// TwinCAT 3 PLC project PLC
// Title: StateFramework
// Company: RoddenLab
// Author: Kevin Rodden
// ProjectVersion: 1.0.0
// Description: Libary for state-based design of PLC software.
// ProgramVersion: 3.1.4023.0
// libraries:
//   Tc2_Standard, * (Beckhoff Automation GmbH)
//   Tc2_System, * (Beckhoff Automation GmbH)
//   Tc2_TcpIp, * (Beckhoff Automation GmbH)
//   Tc2_Utilities, * (Beckhoff Automation GmbH)
//   Tc3_Module, * (Beckhoff Automation GmbH)
// project tree:
//   DUTs/ ComponentIdentifier.TcDUT, DINT100FIFOBuffer.TcDUT, FaultMessage.TcDUT, Framework.TcDUT, FrameworkLocal.TcDUT, GeneralMessage.TcDUT, HMIBanner.TcDUT, HMIMessage.TcDUT, HMIMessageBuffer.TcDUT, ID50FIFOBuffer.TcDUT, LREAL100FIFOBuffer.TcDUT, StateTimeStamp.TcDUT, Station.TcDUT, TraceFIFOBuffer.TcDUT
//   DUTs/Stats/ Component_Stats.TcDUT, StatsAggregateFIFOBuffer.TcDUT, StatsAggregateRecord.TcDUT, StatsConstants.TcDUT, StatsEvent.TcDUT, StatsEventFIFOBuffer.TcDUT, StatsFailure.TcDUT, StatsFailureFIFOBuffer.TcDUT, StatsFault.TcDUT, StatsFaultFIFOBuffer.TcDUT, StatsShiftAggregateFIFOBuffer.TcDUT, StatsShiftAggregateRecord.TcDUT
//   ENUMs/ eChannel.TcDUT, eColor.TcDUT, eRxMode.TcDUT
//   / PlcTask.TcTTO
//   POUs/Framework/ FB_Framework.TcPOU, FB_StationState.TcPOU, FIFO_HMIMessage.TcPOU, F_FindMessage.TcPOU, FB_StationControl.TcPOU
//   POUs/OEE/ FIFO_StatsAggregate.TcPOU, FIFO_StatsEvent.TcPOU, FIFO_StatsFailureLog.TcPOU, FIFO_StatsFaultLog.TcPOU, FIFO_StatsShiftAggregate.TcPOU, F_SendEvent.TcPOU
//   POUs/Serial Communication/ FB_EL6001.TcPOU, FB_EL6002.TcPOU
//   POUs/State Trace/ FIFO_StateTrace.TcPOU
//   POUs/TCP Communication/ FB_TCPClient.TcPOU
//   POUs/Utility/ FB_Blinker.TcPOU, FB_FileReadSettings.TcPOU, FB_FileWriteSettings.TcPOU, FB_Sensor.TcPOU, FIFO_DINT100.TcPOU, FIFO_ID50.TcPOU, FIFO_LREAL100.TcPOU, F_GetTimeStamp.TcPOU, LEFTBigString.TcPOU, RIGHTBigString.TcPOU
// real-time tasks:
//   TASK PlcTask: cycle T#10ms, priority 20, ADS port 350

CONFIGURATION PLC
    RESOURCE PLC ON TwinCAT3
        TASK PlcTask(INTERVAL := T#10ms, PRIORITY := 20);
    END_RESOURCE
END_CONFIGURATION

// ---- DUTs/ComponentIdentifier.TcDUT
TYPE ComponentIdentifier :
STRUCT
	ID		: DINT;		// Component ID
	Name	: STRING;	// Component Name
END_STRUCT
END_TYPE

// ---- DUTs/DINT100FIFOBuffer.TcDUT
TYPE DINT100FIFOBuffer :
STRUCT
	Size	: UDINT := 100;				// Size of FIFO
	Buffer	: ARRAY [0..99] OF DINT;	// Buffer of FIFO Elements
END_STRUCT
END_TYPE

// ---- DUTs/FaultMessage.TcDUT
TYPE FaultMessage :
STRUCT
	Id		: DINT;			// Identifier for Fault Condition
	Text	: T_MaxString;	// Text (Message) for Fault Condition
	AltText	: T_MaxString;	// Alt Text for Fault Condition
END_STRUCT
END_TYPE

// ---- DUTs/Framework.TcDUT
TYPE Framework :
STRUCT
	ComponentIDRecord	: ComponentIdentifier;	// Component Identifier
	Behavior			: DINT;					// Component Behavior Modifier
	OnScan				: BOOL;
	ResetStart			: BOOL;
	ResetDone			: BOOL;
	FullInitRequired	: BOOL;
	EnableStateTrace	: BOOL;
END_STRUCT
END_TYPE

// ---- DUTs/FrameworkLocal.TcDUT
TYPE FrameworkLocal :
STRUCT
	AsynchFault					: BOOL;
	AsynchFaultReactionComplete	: BOOL;
	Attention					: BOOL;
	CycleAuto					: BOOL;
	CycleFaulted				: BOOL;
	CycleManual					: BOOL;
	CycleReset					: BOOL;
	ManualCycleRequested		: BOOL;
	ManualCycleDone				: BOOL;
	OKToStop					: BOOL;
	SingleStepInhibit			: BOOL;
	IgnoreSingleStep			: BOOL;
	FirstEntry					: BOOL;
	LongFaultState				: BOOL;
	CycleAutoFallingEdge		: F_TRIG;
	CycleResetFallingEdge		: F_TRIG;
	CycleManualFallingEdge		: F_TRIG;
	State						: DINT;
	NextState					: DINT;
	LastAutoState				: DINT;
	ReEntryState				: DINT;
	FaultedState				: DINT;
	FaultNumber					: DINT;
	LocalFaultID				: DINT;
	FullFaultID					: DINT;
	tmrState					: TON;
	tmrFault					: TON;
	StateTimePreset				: TIME;
	FaultTimePreset				: TIME;
	FaultTimeLong				: TIME;
	FaultTimeShort				: TIME;
	FaultText					: T_MaxString;
	FaultAltText				: T_MaxString;
	FaultData					: StatsFault;
	MsgText						: T_MaxString;
	AltMsgText					: T_MaxString;
	MsgArray					: ARRAY [0..99] OF GeneralMessage;
	HMIMsg						: HMIMessage;
	StateTimeStamp				: StateTimeStamp;
	CurrentTime					: TimeStamp;
	Name						: STRING(30);
	AltName						: STRING(30);
	pStateTraceBuffer			: POINTER TO TraceFIFOBuffer;
	pStateTraceFifo				: POINTER TO FIFO_StateTrace;
	pStats						: POINTER TO Component_Stats;
END_STRUCT
END_TYPE

// ---- DUTs/GeneralMessage.TcDUT
TYPE GeneralMessage :
STRUCT
	Id: DINT;
	BitNumber: DINT;
	Text: STRING;
	AltText: STRING;
END_STRUCT
END_TYPE

// ---- DUTs/HMIBanner.TcDUT
// HMI Banner Structure Relaying Data to HMI Controls
TYPE HMIBanner :
STRUCT
	Text	: T_MaxString;	// Text for HMI Banner
	AltText	: T_MaxString;	// Additional Text for HMI Banner
	Color	: eColor;		// Color of HMI Banner Background
END_STRUCT
END_TYPE

// ---- DUTs/HMIMessage.TcDUT
TYPE HMIMessage :
STRUCT
	Channel	: eChannel;		// Channel for HMI Message
	Color	: eColor;		// Color of HMI Message (Background)
	Text	: T_MaxString;	// Text of HMI Message
	AltText	: T_MaxString;	// Additional Text for HMI Message
END_STRUCT
END_TYPE

// ---- DUTs/HMIMessageBuffer.TcDUT
TYPE HMIMessageBuffer :
STRUCT
	Size	: UDINT := 100;					// Array Size for HMI Message FIFO Buffer
	Buffer	: ARRAY [0..99] OF HMIMessage;	// FIFO Buffer for HMI Messages 
END_STRUCT
END_TYPE

// ---- DUTs/ID50FIFOBuffer.TcDUT
TYPE ID50FIFOBuffer :
STRUCT
	Size: UDINT := 50;
	Buffer: ARRAY [0..49] OF ComponentIdentifier;
END_STRUCT
END_TYPE

// ---- DUTs/LREAL100FIFOBuffer.TcDUT
TYPE LREAL100FIFOBuffer :
STRUCT
	Size: UDINT := 100;
	Buffer: ARRAY [0..99] OF LREAL;
END_STRUCT
END_TYPE

// ---- DUTs/StateTimeStamp.TcDUT
TYPE StateTimeStamp :
STRUCT
	Station		: DINT;	
	ID			: DINT;
	State		: DINT;
	DateTime	: TIMESTRUCT;
END_STRUCT
END_TYPE

// ---- DUTs/Station.TcDUT
TYPE Station :
STRUCT
	FirstScan					: BOOL	:= TRUE;	// First Scan for PLC Startup
	
	CycleAuto					: BOOL;					// Flag Indicating 
	CycleReset					: BOOL;
	CycleManual					: BOOL;
	CycleStopped				: BOOL;
	CycleFaulted				: BOOL;
	
	OKToStart					: BOOL;					// Flag Indicating Station Readiness to Start Cycling
	OKToStop					: BOOL;					// Flag Indicating Station Readiness to Stop Cycling
	OKToReset					: BOOL;					// Flag Indicating Station Readiness to Reset Faults/Handshakes
	OKForManual					: BOOL;					// Flag Indicating Station Readiness to Enter Manual Mode
	
	StopRequest					: BOOL;
	EmergencyStop				: BOOL;
	UnlatchFaults				: BOOL;
	FaultReset					: BOOL;
	StationResetRequired		: BOOL;					// Flag Indicating Full Station Reset Required
	ResetDone					: BOOL;
	SingleStep					: BOOL;
	StepAdvance					: BOOL;
	DryCycle					: BOOL;
	Attention					: BOOL;
	MachineStopRequest			: BOOL;
	StationID					: DINT;					// Identifier for the Station
	
	FirstFault					: StatsFault;			
	UpstreamStationID			: DINT;					// Upstream Station Identifier
	DownstreamStationID			: DINT;					// Downstream Station Identifier
	
	StationMessage				: HMIBanner;
	OperatorMessage				: HMIBanner;
	b500msPulse					: BOOL;					// Global 500ms Boolean Pulse

	FaultedFIFO					: FIFO_ID50;			// FIFO of Faulted Components
	FaultedFIFOBuffer			: ID50FIFOBuffer;		// Faulted Component FIFO Memory
	
	NotOKtoStopFIFO				: FIFO_ID50;			// FIFO of Not OK to Stop Components
	NotOKToStopFIFOBuffer		: ID50FIFOBuffer;		// Not OK to Stop FIFO Memory
	
	HMIMessageFIFO				: FIFO_HMIMessage;		// FIFO of HMI Messages
	HMIMessageBuffer			: HMIMessageBuffer;		// HMI Message FIFO Memory
	
	AttentionRequiredFIFO		: FIFO_ID50;			// FIFO of Components Requiring Attention
	AttentionRequiredFIFOBuffer	: ID50FIFOBuffer;		// Attention Request FIFO Memory
	
	CycleManualFIFO				: FIFO_ID50;
	CycleManualFIFOBuffer		: ID50FIFOBuffer;
	
	StationStateTraceFifo		: FIFO_StateTrace;
	StationStateTraceBuffer		: TraceFIFOBuffer;	
END_STRUCT
END_TYPE

// ---- DUTs/Stats/Component_Stats.TcDUT
TYPE Component_Stats :
STRUCT
	AggregateInterval			: DINT; 						(*interval time in minutes*)
	PlannedDowntime				: ARRAY [0..2] OF DINT;  		(*index corresponds to shift number*)
	StartOfShift				: ARRAY [0..2, 0..1] OF DINT; 	(*[shift number],[hour,min]*)
	IdealCycleTime				: LREAL; 						(*cycle time is second*)
	StatsEventFIFO				: FIFO_StatsEvent 			:= (Overwrite := TRUE);
	StatsEventBuffer			: StatsEventFIFObuffer;
	StatsAggregateFIFO			: FIFO_StatsAggregate 		:= (Overwrite := TRUE);
	StatsAggregateBuffer		: StatsAggregateFIFOBuffer;
	StatsShiftAggregateFIFO		: FIFO_StatsShiftAggregate 	:= (Overwrite := TRUE);
	StatsShiftAggregateBuffer	: StatsShiftAggregateFIFOBuffer;
	StatsFaultLog				: FIFO_StatsFaultLog 		:= (Overwrite := TRUE);
	StatsFaultLogBuffer			: StatsFaultFIFOBuffer;
	StatsFailureLog				: FIFO_StatsFailureLog 		:= (Overwrite := TRUE);
	StatsFailureLogBuffer		: StatsFailureFIFOBuffer;
	StatsIdealCycleTimeFIFO		: FIFO_LREAL100;
	StatsIdealCycleTimeBuffer	: LREAL100FIFOBuffer;
	StatsPartCountFIFO			: FIFO_DINT100;
	StatsPartCountBuffer		: DINT100FIFOBuffer;
	Framework					: Framework;
END_STRUCT
END_TYPE

// ---- DUTs/Stats/StatsAggregateFIFOBuffer.TcDUT
TYPE StatsAggregateFIFOBuffer :
STRUCT
	Size: UDINT := 864; (*3 days at 5 min*)
	Buffer: ARRAY [0..863] OF StatsAggregateRecord;
END_STRUCT
END_TYPE

// ---- DUTs/Stats/StatsAggregateRecord.TcDUT
TYPE StatsAggregateRecord :
STRUCT
	TimeStamp: TimeStamp;
	OperatorStopTime: LREAL;
	OperatorStopCount: DINT;
	AutoStopTime: LREAL;
	AutoStopCount: DINT;
	WorkTime: LREAL;
	WorkCount: DINT;
	BypassTime: LREAL;
	BypassCount: DINT;
	BlockTime: LREAL;
	BlockCount: DINT;
	StarveTime: LREAL;
	StarveCount: DINT;
	FaultTime: LREAL;
	FaultCount: DINT;
	EmptyTime: LREAL;
	EmptyCount: DINT;
	RetryTime: LREAL;
	RetryCount: DINT;
	MasterTime: LREAL;
	MasterCount: DINT;
	OtherTime: LREAL;
	OtherCount: DINT;
	RejectCount: DINT;
	GoodCount: DINT;
	FirstTimeGoodCount: DINT;
	FirstTimeStartCount: DINT;
	GoodCycleTime: LREAL;
	InitCount: DINT;
	PartsForCurrentCycleTime: DINT;
	Shift: DINT;
END_STRUCT
END_TYPE

// ---- DUTs/Stats/StatsConstants.TcDUT
TYPE StatsConstants :
STRUCT
	Aggregate: DINT := 1;

	OperatorStop: DINT := 100;
	MachineStop: DINT := 101;
	Working: DINT := 102;
	Bypass: DINT := 103;
	Blocked: DINT := 104;
	Starved: DINT := 105;
	Faulted: DINT := 106;
	FaultAcknowledge: DINT := 107;
	Empty: DINT := 108;
	Retry: DINT := 109;
	Mastering: DINT := 110;

	Failure: DINT := 200;
	Good: DINT := 201;
	FirstTimeGood: DINT := 202;
	FirstTimeStart: DINT := 203;
	Initialize: DINT := 204;

	PartChange: DINT := 300;
	CycleTime: DINT := 301;
END_STRUCT
END_TYPE

// ---- DUTs/Stats/StatsEvent.TcDUT
TYPE StatsEvent :
STRUCT
	TimeStamp: TimeStamp;
	EType: DINT;
	Data: ARRAY [0..4] OF REAL;
	StringData: ARRAY [0..3] OF STRING;
END_STRUCT
END_TYPE

// ---- DUTs/Stats/StatsEventFIFOBuffer.TcDUT
TYPE StatsEventFIFOBuffer :
STRUCT
	Size: UDINT := 100;
	Buffer: ARRAY [0..99] OF StatsEvent;
END_STRUCT
END_TYPE

// ---- DUTs/Stats/StatsFailure.TcDUT
TYPE StatsFailure :
STRUCT
	TimeStamp: TimeStamp;
	StationID: DINT;
	FailureID: DINT;
	Parameters: STRING;
END_STRUCT
END_TYPE

// ---- DUTs/Stats/StatsFailureFIFOBuffer.TcDUT
TYPE StatsFailureFIFOBuffer :
STRUCT
	Size: UDINT := 500;
	Buffer: ARRAY [0..499] OF StatsFailure;
END_STRUCT
END_TYPE

// ---- DUTs/Stats/StatsFault.TcDUT
TYPE StatsFault:
STRUCT
	TimeStamp: TimeStamp;
	StationID: DINT;
	FaultID: DINT;
	AcknowledgeTime: LREAL;
	Duration: LREAL;
	Data: ARRAY [0..2] OF REAL;
	StringData: ARRAY [0..3] OF STRING;
END_STRUCT
END_TYPE

// ---- DUTs/Stats/StatsFaultFIFOBuffer.TcDUT
TYPE StatsFaultFIFOBuffer :
STRUCT
	Size: UDINT := 500;
	Buffer: ARRAY [0..499] OF StatsFault;
END_STRUCT
END_TYPE

// ---- DUTs/Stats/StatsShiftAggregateFIFOBuffer.TcDUT
TYPE StatsShiftAggregateFIFOBuffer :
STRUCT
	Size: UDINT := 270; (*90 days*)
	Buffer: ARRAY [0..269] OF StatsShiftAggregateRecord;
END_STRUCT
END_TYPE

// ---- DUTs/Stats/StatsShiftAggregateRecord.TcDUT
TYPE StatsShiftAggregateRecord :
STRUCT
	AggregateData: StatsAggregateRecord;
	Shift: DINT;
	ShiftStartTimeStamp: TimeStamp;
	AvailableTime: LREAL;
	NetAvailableTime: LREAL;
	TotalDownTime: LREAL;
	PlannedDownTime: LREAL;
	UnplannedDownTime: LREAL;
	OperatingTime: LREAL;
	EquipmentAvailability: LREAL;
	TotalParts: DINT;
	PerformanceEfficiency: LREAL;
	QualityRate: LREAL;
	OverallEquipmentEffectiveness: LREAL;
	CycleTimeAvgSum: LREAL;
	CycleTimeAvgCnt: DINT;
END_STRUCT
END_TYPE

// ---- DUTs/TraceFIFOBuffer.TcDUT
TYPE TraceFIFOBuffer :
STRUCT
	Size: UDINT := 1000;
	Buffer: ARRAY [0..999] OF StateTimeStamp;
END_STRUCT
END_TYPE

// ---- ENUMs/eChannel.TcDUT
{attribute 'qualified_only'}
{attribute 'strict'}
TYPE eChannel :
(
	Unspecified	:= 0,	// Message Channel Not Defined
	Fault 		:= 1,	// Fault Channel
	Attention 	:= 2,	// Attention Required Channel
	General 	:= 3,	// General Information Channel
	FirstFault 	:= 4	// First Fault (Startup) Channel
) DINT := Unspecified;
END_TYPE

// ---- ENUMs/eColor.TcDUT
{attribute 'qualified_only'}
{attribute 'strict'}
TYPE eColor :
(
	Black 	:= 16#000000,	// Black RGB Code
	Red	 	:= 16#FF0000,	// Red RGB Code
	Green 	:= 16#00FF00,	// Green RGB Codde
	Blue 	:= 16#0000FF,	// Blue RGB Codee
	Grey 	:= 16#F2F2F2,	// Gray RGB Code
	Yellow 	:= 16#FFFF00,	// Yellow RGB Code
	White 	:= 16#FFFFFF	// White RGB Code
) DINT := Black;
END_TYPE

// ---- ENUMs/eRxMode.TcDUT
{attribute 'qualified_only'}
{attribute 'strict'}
TYPE eRxMode :
(
	Delimited	:= 0,
	FixedLength := 1,
	Continuous	:= 2
);
END_TYPE

// ---- POUs/Framework/FB_Framework.TcPOU
FUNCTION_BLOCK FB_Framework
VAR_INPUT
	ComponentIDRecord	: ComponentIdentifier;	// Information to Identify Component
	CurrentTime			: TimeStamp;			// Current System Time
END_VAR

VAR_IN_OUT
	Local				: FrameworkLocal;		// Framework Local Structure Reference
	Station				: Station;				// Station Object Reference
END_VAR

VAR
	Message				: GeneralMessage;		// Fault Message Memory Buffer
	HMIMessage			: HMIMessage;			// HMI Message Memory Buffer		
END_VAR

// Initialize Framework Local Fields
IF Station.FirstScan THEN
	Local.State 		:= 9999;
	Local.NextState 	:= 5000;
	Local.FaultedState 	:= 0;
	Local.ReEntryState 	:= 0;
	Local.LastAutoState := 0;
	Local.FaultNumber 	:= 0;
END_IF

(****************************************************************************
* Framework Post-Sequence Logic, DO NOT modify this section *
*****************************************************************************)

(****************************************************************************
* State Timeout Fault Logic *
*****************************************************************************)
// Set the State Fault Timer to Preset 
Local.tmrFault(PT := Local.FaultTimePreset);

// If Component in Auto, Reset, or Manual, Fault Enabled
IF Local.CycleAuto OR Local.CycleReset OR Local.CycleManual THEN
	// If Component OK to Stop or Single Stepping, Fault Disabled
	IF NOT Local.OKToStop AND NOT Station.SingleStep THEN
		// If State Stuck for Duration, Trigger Fault
		Local.tmrFault(IN := Local.NextState = Local.State);
	ELSE
		Local.tmrFault(IN := FALSE);
	END_IF
ELSE
	Local.tmrFault(IN := FALSE);
END_IF

// Unlatch Fault Condition When Directed by Station
IF Station.UnlatchFaults THEN
	Local.CycleFaulted := FALSE;
	Local.FaultNumber := 0;
END_IF

// Check if Fault Condition Present
IF Local.FaultNumber > 0 THEN
	
	// If Component not Faulted, Trigger Fault Condition
	IF NOT Local.CycleFaulted THEN
		Local.CycleFaulted := TRUE;
	
		// Check if Fault Occured in Sync with State Machine
		// Set Faulted State/FaultID Accordingly
		IF NOT Local.AsynchFault OR Local.AsynchFaultReactionComplete THEN
			Local.FaultedState := Local.State;
			Local.LocalFaultID := Local.FaultedState * 10 + Local.FaultNumber; // Faulted State Used in Identifier
		ELSE
			Local.FaultedState := 0;
			Local.LocalFaultID := Local.FaultNumber; // No Faulted State Included (Async == Global in this case)
		END_IF
		
		// Set Full Fault ID (Includes Component ID)
		Local.FullFaultID := ComponentIDRecord.ID * 100000 + Local.LocalFaultID;
		Local.FaultData.FaultID := Local.FullFaultID;
		
		// Fetch Message for Fault Condition
		Message := F_FindMessage(Local.MsgArray, Local.FaultedState, Local.FaultNumber);
		
		// Set Local Fault Message Text
		Local.MsgText := 'Fault: ';
		Local.MsgText := CONCAT(Local.MsgText, DINT_TO_STRING(Local.FaultData.FaultID));
		Local.MsgText := CONCAT(Local.MsgText, ' ');
		Local.MsgText := CONCAT(Local.MsgText, Local.Name);
		Local.MsgText := CONCAT(Local.MsgText, ' - ');
		Local.MsgText := CONCAT(Local.MsgText, Message.Text);
		
		// Set Local Alt Fault Message Text
		Local.AltMsgText := 'AltFault: ';
		Local.AltMsgText := CONCAT(Local.AltMsgText, DINT_TO_STRING(Local.FaultData.FaultID));
		Local.AltMsgText := CONCAT(Local.AltMsgText, ' ');
		Local.AltMsgText := CONCAT(Local.AltMsgText, Local.AltName);
		Local.AltMsgText := CONCAT(Local.MsgText, ' - ');
		Local.AltMsgText := CONCAT(Local.AltMsgText, Message.AltText);
		
		// Add Message to Station Buffer
		HMIMessage.Text		:= Message.Text;
		HMIMessage.AltText 	:= Message.AltText;
		HMIMessage.Channel	:= eChannel.Fault;
		HMIMessage.Color	:= eColor.Red;
		Station.HMIMessageFIFO.LOAD(HMIMessage := HMIMessage);
		
		// Check if Component Fault Already Active
		// Set Station First Fault to Current Fault if Not Active
		IF Station.FirstFault.FaultID = 0 THEN
			Station.FirstFault 					:= Local.FaultData;
			Station.FirstFault.StationID 		:= Station.StationID;
			Station.FirstFault.StringData[0] 	:= Local.MsgText;
			Station.FirstFault.StringData[1] 	:= Local.AltMsgText;
			Station.FirstFault.StringData[2] 	:= Local.FaultData.StringData[2];
			Station.FirstFault.Data 			:= Local.FaultData.Data;
		END_IF
	END_IF
END_IF


// If Cycle Faulted, Load Fault to FIFO
IF Local.CycleFaulted THEN
	Station.FaultedFIFO.LOAD(pFIFO := ADR(Station.FaultedFIFOBuffer), In := ComponentIDRecord);
END_IF

// If Cycle Manual, Load Manual to FIFO
IF Local.CycleManual THEN
	Station.CycleManualFIFO.LOAD(pFIFO := ADR(Station.CycleManualFIFOBuffer), in := ComponentIDRecord);
END_IF

// If Attention Flagged, Load to Station FIFO
IF Local.Attention THEN
	Station.AttentionRequiredFIFO.LOAD(pFIFO := ADR(Station.AttentionRequiredFIFOBuffer), in := ComponentIDRecord);
END_IF

// If Not OK to Stop, Load to Station FIFO
IF NOT Local.OKToStop AND NOT Local.CycleFaulted THEN
	Station.NotOKtoStopFIFO.LOAD(pFIFO := ADR(Station.NotOKtoStopFIFOBuffer), in := ComponentIDRecord);
END_IF


(***************************************************************************
* Framework Pre-Sequence Logic, DO NOT modify this section *
****************************************************************************)

// Set Cycle Auto if Station in Auto and Component Not Faulted
Local.CycleAuto := Station.CycleAuto AND NOT Local.CycleFaulted;

// Set Cycle Reset if Station in Reset and Component Not Faulted
Local.CycleReset := Station.CycleReset AND NOT Local.CycleFaulted;

// Set Cycle Manual if Component Requesting Manual and Station Not Faulted
Local.CycleManual := Local.ManualCycleRequested AND NOT Local.ManualCycleDone AND NOT Station.CycleFaulted;

// Set Single Step Mode if Station in Single Step (not Advancing) and Component Enabled
Local.SingleStepInhibit := Station.SingleStep AND NOT Station.StepAdvance AND NOT Local.IgnoreSingleStep;



(*On the falling edge of CycleAuto, grab the current state as LastAutoState.
Also, set the default ReEntryState to the LastAutoState so that we pick back up where we left off after a simple cycle stop / cycle start.
Set State to 5000, the Idle state.
Note that we block the capture of LastAutoState and setting of ReEntryState if we are currently in states 5000 or 5001.
This is to avoid overwriting these values in the rare case that an AsynchFault occurs in the same scans that we are
transitioning out of 5000, or while in 5001.*)
Local.CycleAutoFallingEdge(CLK:=Local.CycleAuto);
IF Local.CycleAutoFallingEdge.Q THEN
	IF Local.State <> 5000 AND Local.State <> 5001 THEN
		Local.LastAutoState := Local.State;
		Local.ReEntryState := Local.LastAutoState;
	END_IF
	Local.NextState := 5000;
END_IF

// On Cycle Reset Falling Edge, Set State to 5000 (Idle)
Local.CycleResetFallingEdge(CLK := Local.CycleReset);
IF Local.CycleResetFallingEdge.Q THEN
	Local.NextState := 5000;
END_IF

// On Manual Cycle Falling Edge, Set State to 5000
Local.CycleManualFallingEdge(Clk:=Local.CycleManual);
IF Local.CycleManualFallingEdge.Q THEN
	Local.NextState := 5000;
END_IF

// On State Transition
IF Local.NextState <> Local.State THEN
	// Set First Entry Flag
	Local.FirstEntry := TRUE;
	
	// Set State Equal to Next State (Update)
	Local.State := Local.NextState;
	
	// Update Current Time
	Local.CurrentTime := CurrentTime;
	
	// Set Data for State Trace Buffer
	Local.StateTimeStamp.ID := ComponentIDRecord.ID;
	Local.StateTimeStamp.State := Local.State;
	Local.StateTimeStamp.DateTime := Local.CurrentTime;
	
	// Add Entry to State Trace Buffer
	Local.pStateTraceFifo^.LOAD(pFIFO := Local.pStateTraceBuffer, IN := Local.StateTimeStamp);
	
ELSE
	// Reset First Entry Flag
	Local.FirstEntry := FALSE;
	
END_IF

// State Idle Timer
Local.tmrState(
	IN := Local.NextState = Local.State,
	PT := Local.StateTimePreset);

// Reset OK to Stop Condition
Local.OKToStop := FALSE;

END_FUNCTION_BLOCK

// ---- POUs/Framework/F_FindMessage.TcPOU
// Function to Retrieve Message from Provided Buffer Mapped to the Provided State/ID Combination
FUNCTION F_FindMessage : GeneralMessage

VAR_INPUT
	MessageArray	: ARRAY [0..99] OF GeneralMessage;	// Array of Messages
	State			: DINT;								// State Reference 
	ID				: DINT;								// Fault ID Reference
END_VAR

VAR
	Message			: GeneralMessage;					// Temporary Message Buffer
	Index			: DINT;								// Index for Array Search
	Length			: DINT;								// Number of Array Elements
END_VAR

// Get Length of Message Array
Length := SIZEOF(MessageArray) / SIZEOF(Message);

// Set Message Text to Defaults
Message.Text 	:= '**No message text**';
Message.AltText := '**No alt message text**';

// Search Message Array for Fault Message
FOR Index := 0 TO (length - 1) DO
	// If Message ID Matches State ID, Set Message Buffer to Array Element
	IF MessageArray[Index].Id = (State * 10 + ID) THEN
		Message := MessageArray[Index];
		EXIT;
	END_IF
END_FOR

// Set Output to Message Buffer
F_FindMessage := Message;

END_FUNCTION

// ---- POUs/Framework/FB_StationState.TcPOU
FUNCTION_BLOCK FB_StationState
// Station State Commands
VAR_INPUT
	StationResetCommand		: BOOL;
	FaultAcknowledgeCommand	: BOOL;
	FaultResetCommand		: BOOL;
	StationLevelFault		: BOOL;
	CycleStartCommand		: BOOL;
	CycleStopCommand		: BOOL;
	ManualModeCommand		: BOOL;
END_VAR

// Configuration Inputs
VAR_INPUT
	SeperateAckAndReset		: BOOL;		// Configuration to Require Fault Acknowledge
	ResetAfterManualMode	: BOOL;		// Configuration to Require Station Reset After Leaving Manual Mode
END_VAR

VAR_IN_OUT
	Station					: Station;
END_VAR

VAR_OUTPUT
	StationStateMessage		: T_MaxString;
END_VAR

VAR
	State					: DINT;
	NextState				: DINT;
	FirstEntry				: BOOL;
	WaitForFaultAck			: BOOL;
	CurrentTime				: TIMESTRUCT;
	ModeTimeStamp			: StateTimeStamp;
END_VAR

// First Scan
IF Station.FirstScan THEN
	State 		:= 9999;
	NextState 	:= 0;
END_IF


// Async Setting for Init Required Flag
IF StationResetCommand THEN
	Station.StationResetRequired := TRUE;
END_IF;


// Mode Control State Machine
CASE State OF
		
	0:	// Faulted, Not Acknowledged
	
		StationStateMessage := 'Faulted, Not Acknowledged';
	
		IF FaultAcknowledgeCommand OR NOT SeperateAckAndReset THEN
			FaultAcknowledgeCommand := FALSE;
			NextState := 10;
		END_IF;
		
	
	10:	// Faulted, Acknowledged
	
		IF FirstEntry THEN
			IF SeperateAckAndReset THEN
				StationStateMessage := 'Fault Acknowledged';
			END_IF;
			WaitForFaultAck := TRUE;
		END_IF;
	
		// Check if Station Ready for Reset
		IF Station.OKToReset THEN
			
			IF WaitForFaultAck AND SeperateAckAndReset THEN
				WaitForFaultAck := FALSE;
				
				IF Station.StationResetRequired THEN
					StationStateMessage := 'Waiting for Station Reset';
				ELSE
					StationStateMessage := 'Waiting for Station or Fault Reset';
				END_IF
			END_IF;
			
			// Check if Station Reset Required
			IF Station.StationResetRequired THEN
				
				// Station Reset Commanded
				IF StationResetCommand THEN
					StationResetCommand 		:= FALSE;
					NextState 			:= 50;
					Station.SingleStep	:= FALSE;
				END_IF
				
				// Fault Reset - Reject
				IF FaultResetCommand THEN
					StationStateMessage := 'Station Reset Required'; 
				END_IF
				
			ELSE
				// Station Reset Commanded
				IF StationResetCommand THEN
					StationResetCommand 		:= FALSE;
					NextState 			:= 50;
					Station.SingleStep	:= FALSE;
				END_IF;
			
				// Fault Reset Commanded
				IF FaultResetCommand THEN
					FaultResetCommand 			:= FALSE;
					NextState  			:= 20;
					Station.SingleStep	:= FALSE;
				END_IF;
			END_IF
			
		END_IF;
		
	
	20	:	// Unlatch Faults, Fault Reset
	
		IF FirstEntry THEN
			Station.UnlatchFaults := TRUE;
			StationStateMessage := 'Unlatching Faults...';
		END_IF;
	
		IF NOT Station.CycleFaulted AND NOT StationLevelFault THEN
			NextState	:= 30;
		END_IF;
	
		IF NextState <> State THEN
			Station.UnlatchFaults := FALSE;
		END_IF
		
		
	30:	// Fault Reset
	
		// Command Component Reset 
		IF FirstEntry THEN
			Station.CycleReset 	:= TRUE;
			StationStateMessage 		:= 'Resetting...';
		END_IF;
	
		// Wait for Reset Complete
		IF Station.ResetDone THEN
			NextState := 100;
		END_IF;
		
		// If Station Faults During Reset or Station Reset Commanded, Return to Faulted
		IF Station.CycleFaulted OR StationResetCommand THEN
			StationResetCommand 	:= FALSE;
			NextState 		:= 0;
		END_IF;
		
		// Reset Component Reset
		IF NextState <> State THEN
			Station.CycleReset := FALSE;
		END_IF
		
	
	50	:	// Unlatch Faults - Station Reset*)
	
		// Unlatch Component Faults
		IF FirstEntry THEN
			Station.UnlatchFaults 	:= TRUE;
			StationStateMessage 			:= 'Unlatching Faults...';
		END_IF;
		
		// Wait for Faults (and Station Faults) to Clear
		IF NOT Station.CycleFaulted AND NOT StationLevelFault THEN
			NextState 	:= 60;
		END_IF;
	
		// Reset Fault Unlatch Command
		IF NextState <> State THEN
			Station.UnlatchFaults	:= FALSE;
		END_IF
		
		
	60	:	// Station Reset
	
		// Command Component Resets
		IF FirstEntry THEN
			Station.CycleReset 	:= TRUE;
			StationStateMessage 		:= 'Resetting...';
		END_IF;
	
		// Wait for Component Reset Complete
		IF Station.ResetDone THEN
			Station.StationResetRequired 	:= FALSE;
			NextState 						:= 100;
		END_IF;
		
		// If Fault During Reset, Return to Faulted State
		IF Station.CycleFaulted THEN
			NextState 	:= 0;
		END_IF;
		
		// Reset Component Reset Command on Exit
		IF NextState <> State THEN
			Station.CycleReset := FALSE;
		END_IF
	
		
	100:	// Idle
	
		IF FirstEntry THEN
			StationStateMessage := 'Idle';
		END_IF
	
		// Cycle Start Commanded
		IF CycleStartCommand AND Station.OKToStart THEN
			CycleStartCommand	:= FALSE;
			NextState 	:= 200;
		END_IF
	
		// Manual Mode Commanded
		IF ManualModeCommand AND Station.OKForManual THEN
			ManualModeCommand	:= FALSE;
			NextState	:= 300;
		END_IF
		
		// In Case of Cycle Fault
		IF Station.CycleFaulted THEN
			NextState := 0;
		END_IF;
		
		// Station Reset Commanded
		IF StationResetCommand AND Station.OKToReset THEN
			NextState := 60;
		END_IF
		
	
	200	:	// Running
	
		IF FirstEntry THEN
			Station.CycleAuto 	:= TRUE;
			StationStateMessage 		:= 'Running';
		END_IF
		
		// Cycle Stop, Operator Stop
		IF CycleStopCommand OR Station.CycleFaulted THEN
			CycleStopCommand	:= FALSE;
			NextState 	:= 250;
		END_IF
	
		
	250 :	// Stop Station
	
		IF FirstEntry THEN
			Station.StopRequest := TRUE;
			StationStateMessage 		:= 'Stopping...';
		END_IF;
		
		// Wait for OK To Stop
		IF Station.OKToStop THEN
			Station.StopRequest := FALSE;
			Station.CycleAuto 	:= FALSE;
			// Check if Fault Occured
			IF Station.CycleFaulted THEN
				NextState := 0;
			ELSE
				NextState := 100;
			END_IF
		END_IF
		
		
	300	:	// Manual Mode
	
		IF FirstEntry THEN
			Station.CycleManual := TRUE;
			StationStateMessage 		:= 'Manual Mode';
		END_IF
		
		// Wait for Stop Command or Fault
		IF CycleStopCommand OR Station.CycleFaulted THEN
			CycleStopCommand := FALSE;
			NextState := 250;
		END_IF
		
		IF State <> NextState THEN
			Station.CycleManual				:= FALSE;
			// Set Station Reset if Configured
			Station.StationResetRequired	:= ResetAfterManualMode;
		END_IF
	
END_CASE


// State Update Logic
IF NextState <> State THEN
	FirstEntry 				:= TRUE;
	State 					:= NextState;
	
	// Update State Trace
	ModeTimeStamp.DateTime	:= F_GetTimeStamp();
	ModeTimeStamp.State		:= NextState;
	ModeTimeStamp.Station	:= Station.StationID;
	Station.StationStateTraceFIFO.LOAD(IN := ModeTimeStamp);
ELSE
	FirstEntry 	:= FALSE;
	
END_IF

END_FUNCTION_BLOCK

// ---- POUs/Utility/F_GetTimeStamp.TcPOU
FUNCTION F_GetTimeStamp : TIMESTRUCT
VAR
	fbGetTime		: GETSYSTEMTIME;	// Function Block to Fetch System Time
	TimeStamp		: T_FileTime;		// Time Stamp Structure
	Time64			: T_ULarge_Integer;	// 64-Bit Large Integer Time
	TimeShift		: LREAL;			// Amount for Time Zone Offset Shift 
	TimeZoneOffset	: DINT;				// UTC Time Zone Offset
END_VAR

// Trigger TwinCAT Function Block
fbGetTime(
	timeLoDW => Time64.dwLowPart, 
	timeHiDW => Time64.dwHighPart);

// Correct for Timezone Offset
TimeShift := DINT_TO_LREAL(ABS(TimeZoneOffset)) (*hours*) * DINT_TO_LREAL(3600) (*seconds*) * DINT_TO_LREAL(10000000) (*100ns*);

IF TimeZoneOffset < 0 THEN
	Time64 := UInt64Sub64(Time64, LREAL_TO_UINT64(TimeShift));
ELSE
	Time64 := UInt64Add64(Time64, LREAL_TO_UINT64(TimeShift));
END_IF

// Unpack Large Integer Time
TimeStamp.dwLowDateTime  := Time64.dwLowPart;
TimeStamp.dwHighDateTime := Time64.dwHighPart;

// Unpack TimeStamp to Time Structure
F_GetTimeStamp :=  FILETIME_TO_SYSTEMTIME(TimeStamp);

END_FUNCTION

// ---- POUs/Framework/FIFO_HMIMessage.TcPOU
// HMI Message FIFO
FUNCTION_BLOCK FIFO_HMIMessage

VAR_INPUT
	Overwrite	: BOOL;							// Flag to Overwrite FIFO Elements (when filled)
	pFIFO		: POINTER TO HMIMessageBuffer;	// Pointer to FIFO Memory
END_VAR

VAR_OUTPUT
	Error		: BOOL;							// Flag Indicating Error with FIFO
	Count		: DINT;							// Count of Elements Within FIFO
	Full		: BOOL;							// Flag Indicating FIFO Full
END_VAR

VAR
	Head		: UDINT;						// Index of Head Element (Newest)
	Tail		: UDINT;						// Index of Tail Element (Oldest)
END_VAR

ACTION INIT:
// Clear Buffer and Output Data
MEMSET(ADR(pFIFO^.Buffer), 0, SIZEOF(pFIFO^.Buffer));

// Reset Count / Indicies
Count 	:= 0;
Head 	:= 0;
Tail 	:= 0;

// Reset Flags
Full 	:= FALSE;
Error 	:= FALSE;
END_ACTION

METHOD LOAD : BOOL
VAR_INPUT
	Input	: HMIMessage;
END_VAR
// Set Success Flag
Error := FALSE;
LOAD := TRUE;

// Check if FIFO Has Room (or Overwrite Enabled)
IF (Full AND Overwrite) OR NOT Full THEN
	
	// Set Head Element to Input Value
	pFIFO^.Buffer[Head] := Input;
	
	// Iterate Head Index
	Head := Head + 1;
	
	// Check if Head at Maximum Value, Rollover
	IF Head = pFIFO^.Size THEN
		Head := 0;
	END_IF
	
	// If FIFO Full, Iterate Tail
	IF Full THEN
		Tail := Tail + 1;
		
		// If Tail at Maximum Value, Rollover
		IF Tail = pFIFO^.Size THEN
			Tail := 0;
		END_IF
		
	// Otherwise Update Count
	ELSE
		Count := Count + 1;
	END_IF
	
// Otherwise, Flag Failure (Value Appended to Full FIFO)
ELSE
	Error := TRUE;
	LOAD := FALSE;
	
END_IF

Full := Head = Tail;
END_METHOD

METHOD PEEK : HMIMessage
// Reset Error Flag
Error := FALSE;

// Check if FIFO Full or Tail
IF Count > 0 THEN
	PEEK := pFIFO^.Buffer[Tail];
	
// Otherwise, Flag Error (FIFO is Empty)
ELSE
	Error := TRUE;
END_IF
END_METHOD

METHOD UNLOAD : HMIMessage
// Reset Error Flag
Error := FALSE;

// Check if FIFO Has Elements
IF Count > 0 THEN
	
	// Fetch Oldest Value from FIFO
	UNLOAD := pFIFO^.Buffer[Tail];
	
	// Clear FIFO Position
	pFIFO^.Buffer[Tail] := 0; 
	
	// Update Oldest Value Index
	Tail := Tail + 1;
	
	// Update Element Count
	Count := Count - 1;
	
	// Check for Rollover
	IF Tail = pFIFO^.Size THEN
		Tail := 0;
	END_IF
	
	// Reset Full Flag
	Full := FALSE;
	
// Otherwise, Flag Error (FIFO is Empty)
ELSE
	Error 	:= TRUE;
	UNLOAD := 0;
END_IF
END_METHOD

END_FUNCTION_BLOCK

// ---- POUs/Framework/FB_StationControl.TcPOU
FUNCTION_BLOCK FB_StationControl

VAR
	Blinker					: FB_Blinker;			// Global 500ms Blinker Function Block
	FaultData				: StatsFault;			// Station Fault Data Statistics
	StationFaultMessage		: HMIMessage;			// Station-Level HMI Message
	tonAirSystemFaultDelay	: TON;					// TON Delay for Air System Fault
	cmdMachineStop			: BOOL; 				// Command to Stop Machine Cycle
	StationLevelFault		: BOOL;					// Flag for Station Level Fault
	FaultNumber				: INT;					// Current Fault Number
	HMIFaultMessage			: HMIMessage;			// HMI Banner Fault Message
	WaitForFaultAck			: BOOL;
	ProcessCompleteTON		: TON;			
END_VAR;

VAR_INPUT
	EmergencyStopStatus		: BOOL;					// Status of Emergency Stop Input
END_VAR

VAR_OUTPUT
	Station					: Station;
END_VAR


VAR_INPUT
	hiCycleStart			: BOOL;
	hiCycleStop				: BOOL;
	hiManualMode			: BOOL;
	hiEstopReset			: BOOL;
	hiFaultAck				: BOOL;
	hiFaultReset			: BOOL;
	hiStationReset			: BOOL;
	hiSingleStepOn			: BOOL;
	hiSingleStepOff			: BOOL;
	hiSingleStep			: BOOL;
	hiDryCycle				: BOOL;
END_VAR

VAR_OUTPUT
	hoOperatorMessage		: STRING;
	hoStationStateMessage	: STRING;
	hoFaultAlert			: BOOL;
	hoOKToStart				: BOOL;
	hoOKToStop				: BOOL;
	hoOKToReset				: BOOL;
END_VAR

// First Scan Initalization ////////////////////////////////////////////////////////////

IF Station.FirstScan THEN
	Station.FirstScan			:= FALSE;
	FaultNumber 				:= 1;
	StationFaultMessage.Text 	:= 'Fault: 1 - PLC First Scan';
	StationFaultMessage.AltText := 'Fault: 1 - PLC First Scan';
	StationFaultMessage.Channel	:= eChannel.FirstFault;
	StationFaultMessage.Color	:= eColor.Red;
	Station.StationID 			:= 10;
END_IF;


// Station Controls

Station.CycleFaulted 	:= StationLevelFault OR Station.FaultedFIFO.Count > 0;
Station.Attention 		:= Station.AttentionRequiredFIFO.Count > 0;

ReadyForManual();
ReadyForStart();
ReadyForStop();
ReadyForReset();

StationState();
SingleStep();


// E-Stop Mode Control Logic ////////////////////////////////////////////////////////////

Station.EmergencyStop := EmergencyStopStatus;

IF Station.EmergencyStop THEN
	IF Station.CycleAuto OR Station.CycleReset OR Station.CycleManual THEN
		FaultNumber 				:= 2;
		StationFaultMessage.Text 	:= 'Fault: 2 - Emergency Stop During Cycle';
		StationFaultMessage.AltText := 'Fault: 2 - Emergency Stop During Cycle';
		StationFaultMessage.Channel	:= eChannel.Fault;
		StationFaultMessage.Color	:= eColor.Red;
	END_IF;
END_IF;


// Station Level Fault Logic ////////////////////////////////////////////////////////////

IF FaultNumber <> 0 AND NOT StationLevelFault THEN
	StationLevelFault 					:= TRUE;
	FaultData.FaultID 					:= FaultNumber;
	Station.FirstFault 					:= FaultData;
	Station.FirstFault.StationID 		:= Station.StationID;
	Station.FirstFault.StringData[0] 	:= StationFaultMessage.Text;
	Station.FirstFault.StringData[1] 	:= StationFaultMessage.AltText;
	
ELSIF Station.UnlatchFaults THEN
	FaultNumber 		:= 0;
	StationLevelFault 	:= FALSE;
	MEMSET(ADR(FaultData), 0, SIZEOF(FaultData));
	MEMSET(ADR(StationFaultMessage), 0, SIZEOF(StationFaultMessage));
	MEMSET(ADR(Station.FirstFault), 0, SIZEOF(Station.FirstFault));
	
END_IF;


// HMI Fault Message Logic

Station.OperatorMessage.Text 	:= Station.FirstFault.StringData[0];
Station.OperatorMessage.Color	:= eColor.Red;

hoOperatorMessage := Station.FirstFault.StringData[0];


// 500ms Station Blinker //////////////////////////////////////////////////////////////////

Blinker(
	IN 	:= TRUE, 
	PT 	:= T#500MS,
	Q	=> Station.b500msPulse);


// Clear Status FIFO Buffers //////////////////////////////////////////////////////////////

Station.AttentionRequiredFIFO.INIT(pFIFO := ADR(Station.AttentionRequiredFIFOBuffer));
Station.NotOKtoStopFIFO.INIT(pFIFO := ADR(Station.NotOKToStopFIFOBuffer));
Station.FaultedFIFO.INIT(pFIFO := ADR(Station.FaultedFIFOBuffer));
Station.CycleManualFIFO.INIT(pFIFO := ADR(Station.CycleManualFIFOBuffer));

// Reset Done

Station.ResetDone := Stn10_10_Main.JRFramework.ResetDone 
	AND Stn10_11_Robot.JRFramework.ResetDone 
	AND Stn10_12_Aligner.JRFramework.ResetDone 
	AND Stn10_13_Laser.JRFramework.ResetDone
	AND Stn10_14_BottomCamera.JRFramework.ResetDone
	AND Stn10_15_TopCamera.JRFramework.ResetDone
	AND Stn10_16_SMIFPodLt.JRFramework.ResetDone
	AND Stn10_17_SMIFPodRt.JRFramework.ResetDone;


// Dry Cycle Enable / Disable Logic
	
IF hiDryCycle AND NOT Station.DryCycle THEN
	hiDryCycle 			:= FALSE;
	Station.DryCycle 	:= TRUE;
	
ELSIF hiDryCycle AND Station.DryCycle THEN
	hiDryCycle 			:= FALSE;
	Station.DryCycle 	:= FALSE;
	
END_IF


// HMI Feedback ///////////////////////////////////////////////

hoFaultAlert 	:= Station.b500msPulse AND Station.CycleFaulted;
hoOKToStart 	:= OKToStart AND NOT Stn10_20_GEM.RemoteModeActive;
hoOKToStop 		:= NOT Stn10_20_GEM.RemoteModeActive OR Station.CycleManual;
hoOKToReset		:= OKToReset;

ACTION ReadyForManual:
Station.OKForManual := NOT Station.CycleAuto 
	AND NOT Station.CycleReset 
	AND NOT Station.StationResetRequired
	AND NOT Station.CycleFaulted
	AND Stn10_11_Robot.APIOut.Connected 
	AND Stn10_12_Aligner.APIOut.Connected
	AND Stn10_13_Laser.APIOut.Connected
	AND Stn10_14_BottomCamera.APIOut.Connected
	AND Stn10_15_TopCamera.APIOut.Connected;
END_ACTION

ACTION ReadyForReset:
OKToReset := NOT Station.EmergencyStop AND NOT Station.CycleManual;
END_ACTION

ACTION ReadyForStart:
OKToStart := NOT Station.EmergencyStop 
	AND NOT Station.CycleFaulted
	AND NOT Station.StationResetRequired 
	AND NOT Station.CycleManual
	AND NOT Station.CycleAuto
	AND Stn10_11_Robot.APIOut.Connected 
	AND Stn10_12_Aligner.APIOut.Connected
	AND Stn10_13_Laser.APIOut.Connected
	AND Stn10_14_BottomCamera.APIOut.Connected
	AND Stn10_15_TopCamera.APIOut.Connected
	AND (NOT F_CassetteEmpty(pMain^.CassetteA) 
		OR NOT F_CassetteEmpty(pSMIFLeft^.Cassette) 
		OR NOT F_CassetteEmpty(pSMIFRight^.Cassette) 
		OR NOT F_CassetteEmpty(pMain^.CassetteB)
		OR Stn10_16_SMIFPodLt.INSTALLED
		OR Stn10_17_SMIFPodRt.INSTALLED)
	AND (Stn10_16_SMIFPodLt.iLeftLoadPlusReady OR NOT Stn10_16_SMIFPodLt.INSTALLED)
	AND (Stn10_17_SMIFPodRt.iRightLoadPlusReady OR NOT Stn10_17_SMIFPodRt.INSTALLED);
END_ACTION

ACTION ReadyForStop:
OKToStop := Station.NotOKtoStopFIFO.Count = 0;
END_ACTION

ACTION SingleStep:
IF hiSingleStepOn THEN
	hiSingleStepOn 		:= FALSE;
	Station.SingleStep 	:= TRUE;
	
ELSIF hiSingleStepOff OR hiStationReset THEN
	hiSingleStepOff		:= FALSE;
	hiStationReset		:= FALSE;
	Station.SingleStep 	:= FALSE;
	
END_IF

IF Station.SingleStep AND hiSingleStep THEN
	hiSingleStep		:= FALSE;
	Station.StepAdvance := TRUE;
ELSE
	Station.StepAdvance := FALSE;	
END_IF
END_ACTION

END_FUNCTION_BLOCK

// ---- POUs/Utility/FB_Blinker.TcPOU
FUNCTION_BLOCK FB_Blinker
VAR_INPUT
	IN	: BOOL;
	PT	: TIME;
END_VAR
VAR_OUTPUT
	Q	: BOOL;
END_VAR
VAR
	TON	: TON;
	TOF	: TOF;
END_VAR

TOF(IN := NOT TON.Q AND IN, PT := PT);
TON(IN := IN AND TOF.Q, PT := PT);

Q := TON.Q;

END_FUNCTION_BLOCK

// ---- POUs/OEE/FIFO_StatsAggregate.TcPOU
FUNCTION_BLOCK FIFO_StatsAggregate
VAR_INPUT
	Overwrite: BOOL;
	pFIFO: POINTER TO StatsAggregateFIFOBuffer;
	in: StatsAggregateRecord;
END_VAR

VAR_OUTPUT
	Err: BOOL;
	Count: DINT;
	Full: BOOL;
	out: StatsAggregateRecord;
END_VAR

VAR
	Head	: UDINT;
	Tail	: UDINT;
	Idx		: UDINT;
END_VAR

ACTION INIT:
Idx := pFIFO^.Size * SIZEOF(in);
MEMSET(ADR(pFIFO^.Buffer[0]), 0, Idx);
MEMSET(ADR(in), 0, SIZEOF(in));
MEMSET(ADR(out), 0, SIZEOF(out));
Count := 0;
Head := 0;
Tail := 0;
Full := 0;
Err := 0;
END_ACTION

ACTION LOAD:
Err := 0;
IF (Full AND Overwrite) OR NOT Full THEN
	pFIFO^.Buffer[Head] := in;
	Head := Head + 1;
	IF Head = pFIFO^.Size THEN
		Head := 0;
	END_IF
	IF Full THEN
		Tail := Tail + 1;
		IF Tail = pFIFO^.Size THEN
			Tail := 0;
		END_IF
	ELSE
		Count := Count + 1;
	END_IF
ELSE
	Err := 1;
END_IF
Full := (Head = Tail);
END_ACTION

ACTION PEEK:
Err := 0;
IF Full OR (Tail <> Head) THEN
	out := pFIFO^.Buffer[Head];
ELSE
	Err := 1; (*fifo is empty*)
END_IF
END_ACTION

ACTION PEEKLAST:
Err := 0;
IF Full OR (Tail <> Head) THEN
	out := pFIFO^.Buffer[Tail];
ELSE
	Err := 1; (*fifo is empty*)
END_IF
END_ACTION

ACTION UNLOAD:
Err := 0;
IF NOT Full AND (Head = Tail) THEN
	(*empty*)
	Err := 1;
ELSE
	out := pFIFO^.Buffer[Tail];
	MEMSET(ADR(pFIFO^.Buffer[Tail]), 0, SIZEOF (in));
	Tail := Tail + 1;
	Count := Count - 1;
	IF Tail = pFIFO^.Size THEN
		Tail := 0;
	END_IF
	Full := 0;
END_IF
END_ACTION

END_FUNCTION_BLOCK

// ---- POUs/OEE/FIFO_StatsEvent.TcPOU
FUNCTION_BLOCK FIFO_StatsEvent
VAR_INPUT
	Overwrite	: BOOL;								// Flag to Overwrite FIFO Elements (when filled)
	pFIFO		: POINTER TO StatsEventFIFOBuffer;	// Pointer to FIFO Memory
END_VAR

VAR_OUTPUT
	Error		: BOOL;								// Flag Indicating Error with FIFO
	Count		: DINT;								// Count of Elements Within FIFO
	Full		: BOOL;								// Flag Indicating FIFO Full
END_VAR

VAR
	Head		: UDINT;							// Index of Head Element (Newest)
	Tail		: UDINT;							// Index of Tail Element (Oldest)
END_VAR

ACTION INIT:
// Clear Buffer and Output Data
MEMSET(ADR(pFIFO^.Buffer), 0, SIZEOF(pFIFO^.Buffer));

// Reset Count / Indicies
Count 	:= 0;
Head 	:= 0;
Tail 	:= 0;

// Reset Flags
Full 	:= FALSE;
Error 	:= FALSE;
END_ACTION

METHOD LOAD : BOOL
VAR_INPUT
	Input	: StatsEvent;
END_VAR
// Set Success Flag
Error := FALSE;
LOAD := TRUE;

// Check if FIFO Has Room (or Overwrite Enabled)
IF (Full AND Overwrite) OR NOT Full THEN
	
	// Set Head Element to Input Value
	pFIFO^.Buffer[Head] := Input;
	
	// Iterate Head Index
	Head := Head + 1;
	
	// Check if Head at Maximum Value, Rollover
	IF Head = pFIFO^.Size THEN
		Head := 0;
	END_IF
	
	// If FIFO Full, Iterate Tail
	IF Full THEN
		Tail := Tail + 1;
		
		// If Tail at Maximum Value, Rollover
		IF Tail = pFIFO^.Size THEN
			Tail := 0;
		END_IF
		
	// Otherwise Update Count
	ELSE
		Count := Count + 1;
	END_IF
	
// Otherwise, Flag Failure (Value Appended to Full FIFO)
ELSE
	Error := TRUE;
	LOAD := FALSE;
	
END_IF

Full := Head = Tail;
END_METHOD

METHOD PEEK : StatsEvent
// Reset Error Flag
Error := FALSE;

// Check if FIFO Full or Tail
IF Count > 0 THEN
	PEEK := pFIFO^.Buffer[Tail];
	
// Otherwise, Flag Error (FIFO is Empty)
ELSE
	Error := TRUE;
END_IF
END_METHOD

METHOD UNLOAD : StatsEvent
// Reset Error Flag
Error := FALSE;

// Check if FIFO Has Elements
IF Count > 0 THEN
	
	// Fetch Oldest Value from FIFO
	UNLOAD := pFIFO^.Buffer[Tail];
	
	// Clear FIFO Position
	pFIFO^.Buffer[Tail] := 0; 
	
	// Update Oldest Value Index
	Tail := Tail + 1;
	
	// Update Element Count
	Count := Count - 1;
	
	// Check for Rollover
	IF Tail = pFIFO^.Size THEN
		Tail := 0;
	END_IF
	
	// Reset Full Flag
	Full := FALSE;
	
// Otherwise, Flag Error (FIFO is Empty)
ELSE
	Error 	:= TRUE;
	UNLOAD := 0;
END_IF
END_METHOD

END_FUNCTION_BLOCK

// ---- POUs/OEE/FIFO_StatsFailureLog.TcPOU
FUNCTION_BLOCK FIFO_StatsFailureLog
VAR_INPUT
	Overwrite: BOOL;
	pFIFO: POINTER TO StatsFailureFIFOBuffer;
	in: StatsFailure;
END_VAR

VAR_OUTPUT
	Err: BOOL;
	Count: DINT;
	Full: BOOL;
	out: StatsFailure;
END_VAR

VAR
	Head: UDINT;
	Tail: UDINT;
	Idx: UDINT;
END_VAR

ACTION INIT:
Idx := pFIFO^.Size * SIZEOF(in);
MEMSET(ADR(pFIFO^.Buffer[0]), 0, Idx);
MEMSET(ADR(in), 0, SIZEOF(in));
MEMSET(ADR(out), 0, SIZEOF(out));
Count := 0;
Head := 0;
Tail := 0;
Full := 0;
Err := 0;
END_ACTION

ACTION LOAD:
Err := 0;
IF (Full AND Overwrite) OR NOT Full THEN
	pFIFO^.Buffer[Head] := in;
	Head := Head + 1;
	IF Head = pFIFO^.Size THEN
		Head := 0;
	END_IF
	IF Full THEN
		Tail := Tail + 1;
		IF Tail = pFIFO^.Size THEN
			Tail := 0;
		END_IF
	ELSE
		Count := Count + 1;
	END_IF
ELSE
	Err := 1;
END_IF
Full := (Head = Tail);
END_ACTION

ACTION PEEK:
Err := 0;
IF Full OR (Tail <> Head) THEN
	out := pFIFO^.Buffer[Tail];
ELSE
	Err := 1; (*fifo is empty*)
END_IF
END_ACTION

ACTION UNLOAD:
Err := 0;
IF NOT Full AND (Head = Tail) THEN
	(*empty*)
	Err := 1;
ELSE
	out := pFIFO^.Buffer[Tail];
	MEMSET(ADR(pFIFO^.Buffer[Tail]), 0, SIZEOF (in));
	Tail := Tail + 1;
	Count := Count - 1;
	IF Tail = pFIFO^.Size THEN
		Tail := 0;
	END_IF
	Full := 0;
END_IF
END_ACTION

END_FUNCTION_BLOCK

// ---- POUs/OEE/FIFO_StatsFaultLog.TcPOU
FUNCTION_BLOCK FIFO_StatsFaultLog
VAR_INPUT
	Overwrite: BOOL;
	pFIFO: POINTER TO StatsFaultFIFOBuffer;
	in: StatsFault;
END_VAR

VAR_OUTPUT
	Err: BOOL;
	Count: DINT;
	Full: BOOL;
	out: StatsFault;
END_VAR

VAR
	Head: UDINT;
	Tail: UDINT;
	Idx: UDINT;
END_VAR

ACTION INIT:
Idx := pFIFO^.Size * SIZEOF(in);
MEMSET(ADR(pFIFO^.Buffer[0]), 0, Idx);
MEMSET(ADR(in), 0, SIZEOF(in));
MEMSET(ADR(out), 0, SIZEOF(out));
Count := 0;
Head := 0;
Tail := 0;
Full := 0;
Err := 0;
END_ACTION

ACTION LOAD:
Err := 0;
IF (Full AND Overwrite) OR NOT Full THEN
	pFIFO^.Buffer[Head] := in;
	Head := Head + 1;
	IF Head = pFIFO^.Size THEN
		Head := 0;
	END_IF
	IF Full THEN
		Tail := Tail + 1;
		IF Tail = pFIFO^.Size THEN
			Tail :=0;
		END_IF
	ELSE
		Count := Count + 1;
	END_IF
ELSE
	Err := 1;
END_IF
Full := (Head = Tail);
END_ACTION

ACTION PEEK:
Err := 0;
IF Full OR (Tail <> Head) THEN
	out := pFIFO^.Buffer[Tail];
ELSE
	Err := 1; (*fifo is empty*)
END_IF
END_ACTION

ACTION UNLOAD:
Err := 0;
IF NOT Full AND (Head = Tail) THEN
	(*empty*)
	Err := 1;
ELSE
	out := pFIFO^.Buffer[Tail];
	MEMSET(ADR(pFIFO^.Buffer[Tail]), 0, SIZEOF (in));
	Tail := Tail + 1;
	Count := Count - 1;
	IF Tail = pFIFO^.Size THEN
		Tail := 0;
	END_IF
	Full := 0;
END_IF
END_ACTION

END_FUNCTION_BLOCK

// ---- POUs/OEE/FIFO_StatsShiftAggregate.TcPOU
FUNCTION_BLOCK FIFO_StatsShiftAggregate
VAR_INPUT
	Overwrite: BOOL;
	pFIFO: POINTER TO StatsShiftAggregateFIFOBuffer;
	in: StatsShiftAggregateRecord;
	PeekCnt: UDINT;
END_VAR

VAR_OUTPUT
	Err: BOOL;
	Count: DINT;
	Full: BOOL;
	out: StatsShiftAggregateRecord;
END_VAR

VAR
	Head: UDINT;
	Tail: UDINT;
	Idx: UDINT;

	PeekHead: UDINT;
	PeekTail: UDINT;
END_VAR

ACTION INIT:
Idx := pFIFO^.Size * SIZEOF(in);
MEMSET(ADR(pFIFO^.Buffer[0]), 0, Idx);
MEMSET(ADR(in), 0, SIZEOF(in));
MEMSET(ADR(out), 0, SIZEOF(out));
Count := 0;
Head := 0;
Tail := 0;
Full := 0;
Err := 0;
END_ACTION

ACTION LOAD:
Err := 0;
IF (Full AND Overwrite) OR NOT Full THEN
	pFIFO^.Buffer[Head] := in;
	Head := Head + 1;
	IF Head = pFIFO^.Size THEN
		Head := 0;
	END_IF
	IF Full THEN
		Tail := Tail + 1;
		IF Tail = pFIFO^.Size THEN
			Tail := 0;
		END_IF
	ELSE
		Count := Count + 1;
	END_IF
ELSE
	Err := 1;
END_IF
Full := (Head = Tail);
END_ACTION

ACTION PEEK:
Err := 0;
PeekHead := Head;
PeekTail := Tail;
FOR Idx := 0 TO PeekCnt DO

	IF NOT Full AND (PeekHead = PeekTail) THEN
		(*empty*)
		Err := 1;
	ELSE
		out := pFIFO^.Buffer[PeekTail];
		PeekTail := PeekTail + 1;

		IF PeekTail = pFIFO^.Size THEN
			PeekTail := 0;
		END_IF
		Full := 0;
	END_IF
END_FOR

PeekCnt := 0;
END_ACTION

ACTION UNLOAD:
Err := 0;
IF NOT Full AND (Head = Tail) THEN
	(*empty*)
	Err := 1;
ELSE
	out := pFIFO^.Buffer[Tail];
	MEMSET(ADR(pFIFO^.Buffer[Tail]), 0, SIZEOF (in));
	Tail := Tail + 1;
	Count := Count - 1;
	IF Tail = pFIFO^.Size THEN
		Tail := 0;
	END_IF
	Full := 0;
END_IF
END_ACTION

END_FUNCTION_BLOCK

// ---- POUs/OEE/F_SendEvent.TcPOU
FUNCTION F_SendEvent : BOOL

VAR_INPUT
	Event			: StatsEvent;
END_VAR

VAR_IN_OUT
	StatsFIFO		: FIFO_StatsEvent;
	Buffer			: StatsEventFIFOBuffer;
END_VAR

VAR
	TempEvent		: StatsEvent;
END_VAR

VAR_EXTERNAL
	gCurrentTime	: TimeStamp;	// Global System Time Variable
END_VAR

// Use Temp Event, Update TimeStamp
TempEvent := Event;
TempEvent.TimeStamp := gCurrentTime;

// Load Event to Stats FIFO
StatsFIFO(pFIFO := ADR(Buffer));
StatsFIFO.LOAD(Input := TempEvent);

END_FUNCTION

// ---- POUs/Serial Communication/FB_EL6001.TcPOU
// Function Block Used to Integrate the EL6001 Serial Communication Card
FUNCTION_BLOCK FB_EL6001
// Control/Integration Inputs
VAR_INPUT
	TransmitBuffer		: ARRAY [0..1023] OF USINT;	// Tx Message Buffer to Remote Connection
	TransmitLength		: UDINT;					// Length of Tx Message
	TransmitData		: BOOL;						// Command to Trigger Message Send
	ReceiveData			: BOOL;						// Command to Trigger Message Receive
	Initialize			: BOOL;						// Command to Initialize Serial Connection
END_VAR

// Configuration Inputs
VAR_INPUT
	Mode				: eRxMode;			// Method for Receiving Messages from Remote
	EOFArray			: ARRAY [0..11] OF USINT;	// Buffer for Message Delimiter
	EOFLength			: UDINT;					// Length of Message Delimiter
	FixedMessageLength	: UDINT;					// Fixed Message Length (for Fixed Length Mode)
END_VAR

// EL6001 Device Connections
VAR
	InData		AT %I* 	: ARRAY [0..22] OF BYTE;	// Input Data from EL6001 Device
	OutData		AT %Q* 	: ARRAY [0..22] OF BYTE;	// Output Data to EL6001 Device
	SW			AT %I*	: UINT;						// Status Word from EL6001 Device
	CW			AT %Q*	: UINT;						// Control Word to EL6001 Device
END_VAR

// Outputs
VAR_OUTPUT
	ReceiveBuffer		: ARRAY [0..1023] OF USINT;	// Rx Message from Remote Connection
	ReceiveLength		: UDINT;						// Length of Rx Message
	DataAvailable		: BOOL;						// Flag Indicating New Rx Data Available
	TransmitComplete	: BOOL;						// Flag Indicating Tx Send Complete
	InitializeComplete	: BOOL;						// Flag Indicating Initialization Completed
	ErrorCode			: DINT;						// Error Code for Exceptions
	Error				: BOOL;						// Flag Indicating Error Condition
END_VAR

// Internal State Machine Variables
VAR
	State				: DINT;						// Current State of Transmission State Machine
	NextState			: DINT;						// Next State (for Exit/Entry Conditions)
	FirstEntry			: BOOL;						// Flag Inicating First Entry to State
	StateDwellTimer		: TON;						// TON to Track State Dwell
	StateTimePreset		: TIME;						// Time Preset for State Dwell Timer
END_VAR

// Internal Memory Buffers
VAR
	NextCW				: UINT;						// Memory for Future CW
	LastSW				: UINT;						// Memory for Previous SW
	InBuffer			: ARRAY [0..1023] OF USINT;	// Buffer for Rx Data
	InBufferDataLength	: UDINT;					// Length of Data in Rx Buffer
	OutBuffer			: ARRAY [0..1023] OF USINT;	// Buffer for Tx Data
	OutBufferDataLength	: UDINT;					// Length of Data in Tx Buffer
	TempBuffer			: ARRAY [0..1023] OF USINT;	// Buffer Used for Bit-Wise Operations
END_VAR

// Internal Flags/Counters
VAR
	GetCharNum			: UDINT;
	SendCharNum			: UDINT;
	TempCW				: DWORD;
	BitIndex			: SINT;
	EOFIndex			: UDINT;
	EOFCount			: UDINT;
	Index				: UDINT;
	SendIndex			: UDINT;
END_VAR

// State Machine Update Logic

IF NextState <> State THEN
	// Set First Entry Flag
	FirstEntry := TRUE;
	
	// Update State to Next State
	State := NextState;
	
	// Clear State Dwell Timer
	StateDwellTimer(IN := FALSE); 
ELSE
	// Reset First Entry Flag
	FirstEntry := FALSE;	
	
	// Start State Dwell Timer
	StateDwellTimer(IN := TRUE, PT := StateTimePreset); 
END_IF


(**********************
* Sequence logic *
***********************)

CASE State OF

0:	// Dispatch

	// Initialize Serial Interface
	IF Initialize THEN
		NextState := 10;
	END_IF
	
	IF NOT Error AND NOT ReceiveData THEN
		// Data from Remote Detected
		IF (SW.1 AND NOT LastSW.1) OR (NOT SW.1 AND LastSW.1) THEN
			NextState := 100;
		END_IF
	END_IF
	
	// Receive Data from RxBuffer
	IF ReceiveData THEN
		NextState := 200;
	END_IF
	
	// Data Not Finished Sending, Resume Send
	IF OutBufferDataLength - SendIndex <> 0 THEN
		NextState := 310;
		
	// New Send Commanded, Trigger Send
	ELSIF TransmitData THEN
		NextState := 300;
	END_IF

	
10:	(*Initialize device*)

	IF FirstEntry THEN
		Error := FALSE;
		ErrorCode := 0;
		NextCW.2 := 1;
	END_IF
	
	StateTimePreset := T#5S;
		
	IF SW.2 THEN
		NextCW.2 := 0;
		NextState := 20;
	END_IF

	// Check for Dwell Error
	IF StateDwellTimer.Q THEN
		Error := TRUE;
		ErrorCode := 4;
		NextCW.2 := 0;
		NextState := 0;
	END_IF

20: 	(*wait for signal to go low*)

	StateTimePreset := T#5S;

	IF NOT SW.2 THEN
		NextState := 30;
	END_IF

	// Check for Dwell Error
	IF StateDwellTimer.Q THEN
		Error := TRUE;
		ErrorCode := 4;
		NextState := 0;
	END_IF

30: // Clear Data

	IF FirstEntry THEN
		// Reset Data Buffers
		MEMSET(ADR(InBuffer), 0, SIZEOF(InBuffer));
		MEMSET(ADR(OutBuffer), 0, SIZEOF(OutBuffer));
		MEMSET(ADR(ReceiveBuffer), 0, SIZEOF(ReceiveBuffer));
		
		// Reset Send/Receive Info
		InBufferDataLength 	:= 0;
		OutBufferDataLength := 0;
		SendIndex 			:= 0;
		SendCharNum 		:= 0;
		NextCW 				:= 0;
		
		// Reset External Handshakes
		ErrorCode 			:= 0;
		Error 				:= FALSE;
		DataAvailable 		:= FALSE;
		TransmitComplete 	:= FALSE;
		InitializeComplete 	:= TRUE;
	END_IF
	
	// Wait for Initialize Handshake Reset
	IF NOT Initialize THEN
		InitializeComplete := FALSE;
		// Return to Dispatch
		NextState := 0;
	END_IF

100: // Fetch Data from Device

	FOR BitIndex := 8 TO 15 DO
		GetCharNum := DWORD_TO_UDINT(CSETBIT32(UDINT_TO_DWORD(GetCharNum), (BitIndex - 8), GETBIT32(SW, BitIndex)));
	END_FOR;
	
	// If Data Fits in RxBuffer, Receive
	IF (InBufferDataLength + GetCharNum) <= SIZEOF(Inbuffer) THEN
		// Copy Input Data to RxBuffer, Starting at Next Entry
		MEMCPY(ADR(InBuffer[InBufferDataLength]), ADR(InData), GetCharNum);
		
		// Extend Input Data Length by Char Num
		InBufferDataLength := InBufferDataLength + GetCharNum;
		
		NextCW.1 := NOT(CW.1);
		
		NextState := 110;
		
	// Data Larger than RxBuffer, Set Error
	ELSE
		Error := TRUE;
		ErrorCode := 1;
		NextState := 0;
	END_IF

110: // Search for Message in Buffer

	// Check Message Mode
	CASE Mode OF
		
		// Delimiter Message Mode
		eRxMode.Delimited:
			
			// Check if Data Available Flag Set (i.e. Message Defined)
			IF NOT DataAvailable THEN
	
				// Cover for Duplicate Character Case ([DD] instead of [D])
				EOFCount := 0;
				
				// Search for Delimiter, Start at Tail and Move to Head
				FOR Index := 0 TO InBufferDataLength - 1 DO
					// Message Delimiter Found
					IF InBuffer[index] = EOFArray[EOFCount] THEN
						EOFCount := EOFCount + 1;
						IF EOFCount = EOFLength THEN
							EOFIndex := Index - EOFLength + 1;
							EXIT;
						END_IF
					ELSE
						IF EOFCount > 0 THEN
							// Reset EOF Counter, Look for New Match
							EOFCount := 0; 
							// Check if Current Index Matches EOF
							IF InBuffer[index] = EOFArray[EOFCount] THEN
								EOFCount := 1;
							END_IF
						END_IF
					END_IF
				END_FOR;
			END_IF
			
			// Delimiter Found in Buffer, Message Defined
			IF EOFIndex > 0 THEN
				// Copy Message up to but not Including Delimiter to Receive Buffer
				MEMCPY(ADR(ReceiveBuffer), ADR(InBuffer[0]), (EOFIndex));
				Index := EOFIndex + EOFLength;
				ReceiveLength := EOFIndex ;
				
				// Check if Data Remaining in Input Buffer
				IF Index < InBufferDataLength THEN
					// Bit-Shift Data to Head of Buffer
					MEMCPY(ADR(TempBuffer[0]), ADR(InBuffer[Index]), (InBufferDataLength-Index));
					MEMSET(ADR(InBuffer), 0, SIZEOF(InBuffer));
					InBufferDataLength := InBufferDataLength - Index;
					MEMCPY(ADR(InBuffer[0]), ADR(TempBuffer[0]), InBufferDataLength);
					
				// Clear Input Buffer
				ELSE
					MEMSET(ADR(InBuffer), 0, SIZEOF(InBuffer));
					InBufferDataLength := 0;
				END_IF
				
				// Set Data Available Flag
				DataAvailable := TRUE;
				EOFIndex := 0;
				
			END_IF
			
			// Return to Dispatch
			NextState := 0;

			
		// Fixed Message Mode
		eRxMode.FixedLength:
			
			// If Input Data Larger than Fixed Length, Copy to Receive Buffer
			IF NOT DataAvailable AND (InBufferDataLength >= FixedMessageLength) THEN
				// Copy to Receive Buffer
				MEMCPY(ADR(ReceiveBuffer), ADR(InBuffer[0]), FixedMessageLength);
				ReceiveLength := FixedMessageLength;
				
				// Remove Message from Input Buffer
				InBufferDataLength := InBufferDataLength - FixedMessageLength;
				
				// Check if Data Still in Input Buffer
				IF InBufferDataLength > 0 THEN
					// Bit-Shift Remaining Data to Buffer Head 
					MEMCPY(ADR(TempBuffer[0]), ADR(InBuffer[FixedMessageLength]), InBufferDataLength);
					MEMSET(ADR(InBuffer), 0, SIZEOF(InBuffer));
					MEMCPY(ADR(InBuffer[0]), ADR(TempBuffer[0]), InBufferDataLength);
					
				// Clear Input Buffer
				ELSE
					MEMSET(ADR(InBuffer), 0, SIZEOF(InBuffer));
					InBufferDataLength := 0;
				END_IF
				
				// Set Data Available Flag
				DataAvailable := TRUE;
			END_IF
			
			// Return to Dispatch
			NextState := 0;

			
		// Continuous Read Mode
		eRxMode.Continuous:
		
			// Return to Dispatch
			NextState := 0;
			
		// Mode Not Defined
		ELSE
			Error := TRUE;
			ErrorCode := 9;
			NextState := 0;
	END_CASE;

	
	
	
200: // Message Received

	IF FirstEntry THEN
		DataAvailable := FALSE;
		MEMSET(ADR(ReceiveBuffer), 0, SIZEOF(ReceiveBuffer));
		ReceiveLength := 0;
		NextState := 0;
	END_IF
	
	// Check if Additional Input Data
	// Proceed to Receive Data 
	IF InBufferDataLength > 0 THEN
		NextState := 110;
		
	// Return to Dispatch
	ELSE
		NextState := 0;
	END_IF


300: // Transmit Message

	IF FirstEntry THEN
		OutBufferDataLength := TransmitLength;
		MEMCPY(ADR(OutBuffer), ADR(TransmitBuffer), TransmitLength);
		SendIndex := 0;
	END_IF
	
	NextState := 310;
	

310: // Send Data to Remote Device

	IF FirstEntry THEN
		// Check if Transmit Data Length Larger than Output Data Buffer
		// Send up to 22 Bytes of Data
		IF OutBufferDataLength - SendIndex > 22 THEN
			SendCharNum := 22;
			MEMCPY(ADR(OutData), ADR(OutBuffer[SendIndex]), SendCharNum);
			SendIndex := SendIndex + 22;
		// Send Remaining Bytes of Data
		ELSE
			SendCharNum := OutBufferDataLength - SendIndex;
			MEMCPY(ADR(OutData), ADR(OutBuffer[SendIndex]), SendCharNum);
			SendIndex := OutBufferDataLength;
		END_IF
		
		NextCW.0 := NOT(CW.0);
	END_IF
	
	StateTimePreset := T#1S;
	
	IF LastSW.0 <> SW.0 THEN
		// Check if All Data Sent
		IF OutBufferDataLength - SendIndex = 0 THEN
			// Proceed to Tranmit Done
			NextState := 320;
		ELSE
			// Return to Dispatch
			NextState := 0;
		END_IF
	END_IF
	
	// Check if Transmit Timeout
	IF StateDwellTimer.Q THEN
		Error := TRUE;
		ErrorCode := 4;
		NextState := 0;
	END_IF

320: // Transmit Done

	// Set Transmit Complete Flag
	IF FirstEntry THEN
		TransmitComplete := TRUE;
	END_IF
	
	// Wait for Transmit Command to Reset
	IF NOT TransmitData THEN
		TransmitComplete := FALSE;
		// Return to Dispatch
		NextState := 0;
	END_IF

END_CASE


(*set output device bits*)
LastSW := SW;
TempCW := NextCW;
FOR BitIndex := 8 TO 15 DO
	TempCW := CSETBIT32(TempCW, (BitIndex ), GETBIT32(SendCharNum,(BitIndex-8)));
END_FOR;
CW := DWORD_TO_UINT(TempCW);

END_FUNCTION_BLOCK

// ---- POUs/Serial Communication/FB_EL6002.TcPOU
FUNCTION_BLOCK FB_EL6002
VAR_INPUT
	pTransmitBuffer	 	: POINTER TO ARRAY [0..cSerialArraySize-1] OF USINT;
	TransmitLength 	 	: DINT;
	pEOF				: POINTER TO ARRAY[0..11] OF USINT;
	EOFLength			: DINT;
	FixedMessageLength	: DINT;
	pReceiveBuffer		: POINTER TO ARRAY [0..cSerialArraySize-1] OF USINT;
	ReceiveData			: BOOL;
	Initialize			: BOOL;
	bVarSize			: BOOL;
END_VAR

VAR_IN_OUT
	iRS232InData 	: ARRAY [0..21] OF SINT;
	iRS232SW 		: UINT;
	oRS232OutData 	: ARRAY [0..21] OF SINT;
	oRS232CW 		: UINT;
END_VAR

VAR_OUTPUT
	ReceiveLength		: DINT;
	DataAvailable		: BOOL;
	Transmitting		: BOOL;
	InitializeComplete	: BOOL;
	ErrorCode			: DINT;
	Error				: BOOL;
	EOFResult			: STRING(256);
END_VAR

VAR
	TransmitState 		: DINT;
	TransmitNextState	: DINT;
	TransmitTimer	 	: TON;
	state: DINT;
	NextState: DINT;
	FirstEntry: BOOL;
	NoFault: BOOL;
	LongFaultState:BOOL;
	FaultTimer: TON;
	FaultTimerDone:BOOL;
	FaultTimerPreset:TIME;
	FaultedState: DINT;
	FaultNumber: DINT;
	FaultText:STRING256;
	FaultAltText:STRING256;
	FaultMsg: FaultMessage;
	LocalFaultID:DINT;
	FullFaultID:DINT;
	MsgText: STRING256;
	AltMsgText:STRING256;
	tmrState:TON;

	LastSW:UINT;
	InBuffer:ARRAY [0..cSerialArraySize-1] OF USINT;
	TempBuffer:ARRAY[0..cSerialArraySize-1] OF USINT;
	TempXBuffer:ARRAY[0..cSerialArraySize-1] OF USINT;
	InBufferDataLength:DINT;
	pInBuffer:POINTER TO STRING(cSerialArraySize);
	OutBuffer:ARRAY [0..cSerialArraySize-1] OF USINT;
	OutBufferDataLength:DINT;
	DevInDataLength:DINT;
	DevOutDataLength:DINT;
	PreviousInMessageLength:DINT;
	
	GetCharNum:UINT;
	SendCharNum:UINT;
	TempCW:UINT;
	Mode:DINT;
	BitIndex :SINT;
	EOFIndex:DINT;
	EOFFound : BOOL;
	Index:DINT;
	SendIndex:DINT := 0;
	FindState:DINT;
	TransmitActive : BOOL;

	rbTemp:DINT;
	OutBufferDataLenth: BOOL;

	TenpCwAfterShift: UINT;
	
	tmrReceive: TON;
	
END_VAR

VAR CONSTANT
	cDevBufferSize 		: DINT 	:= 22;
	cEOF 				: DINT 	:= 1;
	cFixedLength 		: DINT 	:= 2;
	cContinuous 		: DINT 	:= 3;
	cVarSize 			: DINT	:= 4;
	cSerialArraySize	: UINT 	:= 2000;	// Calling moudle must have same sized array pointers passed in.
END_VAR

// Modified by Roy Coffman 11-Jul-2017
//   Changed Var_In   "pMessageEOF"  to just "pEOF"
//   Changed Var_In   "MessageLength" to "FixedMessageLength"
//   Added constant for internal buffer array sizes

IF NextState <> state THEN
	(*code: Log state change into buffer*)
	FirstEntry := TRUE;
	state := NextState;
	tmrState(IN:=FALSE); (*clear timer if state changes*)
ELSE
	FirstEntry := FALSE;
END_IF

IF TransmitNextState <> TransmitState THEN
	TransmitState := TransmitNextState;
END_IF

IF EOFLength > 0 THEN
	Mode := cEOF;
ELSIF FixedMessageLength > 0 THEN
	Mode := cFixedLength;
ELSIF bVarSize THEN
	Mode := cVarSize;
ELSE
	Mode := cContinuous;
END_IF

rbTemp := SIZEOF(pReceiveBuffer^);

(**********************
* Receive Logic     *
***********************)
(* 1. The terminal indicates that there is new data in the process image by changing the state of the “Receive Request” bit SW.1.
   2. The number of bytes received is written in “Input length” SW.7-15.
   3. The controller acknowledges acceptance of the bytes by changing the state of “Receive request” SW.1. *)
// Modified by Roy Coffman 03-Aug-2017
//  Module appears to want ack to match req, not just change state... so set ack = req

IF NOT Error THEN
	IF (InBufferDataLength + 22) < cSerialArraySize THEN (*data will fit in buffer*)
		IF (iRS232SW.1 XOR LastSW.1) THEN
			GetCharNum := SHR(iRS232SW,8);  // Shift the input length, Bit7 - 15 to an INT
			MEMCPY(ADR(InBuffer[InBufferDataLength]),ADR(iRS232InData),GetCharNum);
			InBufferDataLength := InBufferDataLength + GetCharNum;
			oRS232CW.1 := iRS232SW.1;
		END_IF
		//  Note: data analyzed for EOF in state 100 below.
	ELSE
		MEMSET(ADR(InBuffer),0,SIZEOF(InBuffer));
		InBufferDataLength := 0;
		Error := TRUE;
		ErrorCode := 5;
	END_IF	
END_IF

(**********************
* Transmit Logic     *
***********************)
IF TransmitLength > 0 THEN
	// Comment by Roy Coffman... the next mem copy seems wrong using some offset into the data being asked to be
	//   written by the upper level comnponent.   Is the "OutBufferDataLength" suppose to be in the first argument?
	//   This will function as long as OutBufferDataLength = 0 when this code is evaluated.
	// MEMCPY(ADR(OutBuffer),ADR(pTransmitBuffer^[OutBufferDataLength]),DINT_TO_UDINT(TransmitLength)); // Copy transmit buffer into output buffer
	// Made the change 1/5/21 JCG
	MEMCPY(ADR(OutBuffer[OutBufferDataLength]),pTransmitBuffer,DINT_TO_UDINT(TransmitLength)); // Copy transmit buffer into output buffer
	MEMSET(pTransmitBuffer,0,DINT_TO_UDINT(TransmitLength));  // Clear the transmit buffer
	OutBufferDataLength := OutBufferDataLength + TransmitLength;  // Update the output length
	TransmitLength := 0;
END_IF

(* 1. Set “Output length” to char count
   2. Fill “Data Out 0” to “Data Out n” with user data
   3. Change the state of “Transmit request”
   4. The terminal acknowledges receipt of the data by changing the state of the “Transmit accepted” bit.  *)

TransmitTimer(IN:=TransmitState = 10, PT:=T#1S);
CASE TransmitState OF

0:
	IF NOT Initialize AND OutBufferDataLength > 0 THEN (*Have data to send*)
		IF OutBufferDataLength  > 22 THEN
			SendCharNum:=22;
		ELSE
			SendCharNum :=DINT_TO_UINT( OutBufferDataLength);
		END_IF
		MEMSET(ADR(oRS232OutData),0,22);  // Clear the output data
		MEMCPY(ADR(oRS232OutData),ADR(OutBuffer[0]),SendCharNum); (*copy up to 22 chars to device*)
		TempCW := SHL(SendCharNum,8);  // was 8 bit shift 1/5/21 JCG
		TenpCwAfterShift := TempCW;
		oRS232CW := UINT_TO_WORD(oRS232CW) OR UINT_TO_WORD(TempCW);
		oRS232CW.0 := NOT(oRS232CW.0);
		TransmitNextState:=10;
		Transmitting := TRUE;
	ELSE
		Transmitting := FALSE;
	END_IF

10:
	IF iRS232SW.0 XOR LastSW.0 THEN  // Cneck Transmit Accepted bit
		LastSW.0 := iRS232SW.0;
		TempCW := 255;
		oRS232CW := UINT_TO_WORD(oRS232CW) AND UINT_TO_WORD(TempCW);  // Clear the Output Length field  Upper 8 bits
		MEMSET(ADR(TempXBuffer),0,SIZEOF(TempXBuffer));  // Clear the temp buffer
		MEMCPY(ADR(TempXBuffer[0]),ADR(OutBuffer[SendCharNum]),SIZEOF(OutBuffer)-SendCharNum);  // Copy the remaining chars from Out Buffer to temp
		MEMSET(ADR(outbuffer),0,SIZEOF(outbuffer));  // Clear the Out Buffer
		MEMCPY(ADR(OutBuffer),ADR(TempXBuffer),SIZEOF(TempXBuffer));  // Copy the temp back to out buffer
		OutBufferDataLength := OutBufferDataLength - SendCharNum;  // Update the remaining data length
		TransmitNextState := 0;
	END_IF
	IF TransmitTimer.Q THEN
		Error:=TRUE;
		ErrorCode:=4;
		TransmitNextState := 20;
	END_IF

20:
	(*Error*)
	IF Initialize THEN
		TransmitNextState := 0;
	END_IF

END_CASE


(**********************
* Sequence logic  *
***********************)

CASE state OF

0:	(*Wait for command *)

	IF Initialize THEN
		NextState := 10;
	ELSIF InBufferDataLength >0 AND NOT DataAvailable THEN  // Data available in the buffer
		NextState := 100;
	ELSIF ReceiveData THEN
		NextState:=200;
	END_IF

10:	(*Initialize device
   1. Set “Init request” to 1
   2. The terminal confirms successful initialization by setting “Init accepted”
   3. Reset “Init request”
   4. The terminal sets “Init accepted” to 0. *)
   
	IF  FirstEntry THEN
		Error:=0;
		ErrorCode:=0;
		oRS232CW.2 := 1;  // Init Device
		tmrReceive(IN:=FALSE);
	END_IF
	tmrState(In:=TRUE, PT:=t#5s);
	IF iRS232SW.2 THEN  // Init Accepted = on
		// Set trnasmit req and receive ack to zero while initializing module
		//   resets added by Roy Coffman 3-Sug-2017
		oRS232CW.0 := 0;
		oRS232CW.1 := 0;
		oRS232CW.2 := 0;
		NextState:=20;
	END_IF

	IF tmrState.Q THEN
		(*error*)
		Error:=1;
		ErrorCode:=4;
		oRS232CW.2 := 0;
		NextState := 0;
	END_IF

20: 	(*wait for signal to go low*)

	tmrState(In:=TRUE, PT:=t#5s);

	IF NOT iRS232SW.2 THEN  // Init Accepted = off
		NextState:=30;
	END_IF

	IF tmrState.Q THEN
		(*error*)
		Error:=1;
		ErrorCode:=4;
		NextState := 0;
	END_IF

30: 	(*clear data*)

	IF  FirstEntry THEN
		MEMSET( ADR(InBuffer),0,SIZEOF(InBuffer));
		MEMSET(ADR(OutBuffer),0,SIZEOF(OutBuffer));
		MEMSET(pTransmitBuffer,0,SIZEOF(pTransmitBuffer^));
		MEMSET(pReceiveBuffer,0,SIZEOF(pReceiveBuffer^));
		MEMSET(ADR(oRS232OutData), 0, SIZEOF(oRS232OutData));
		MEMSET(ADR(oRS232CW), 0, SIZEOF(oRS232CW));
		InBufferDataLength:=0;
		OutBufferDataLength:=0;
		SendIndex:=0;
		SendCharNum:=0;
		ErrorCode:=0;
		Error:=0;
		DataAvailable:=0;
		InitializeComplete:=1;
	END_IF
	IF NOT Initialize THEN
		InitializeComplete:=0;  // Finish the handshake
		NextState:=0;
	END_IF

100:	(*Search for message*)

	CASE Mode OF

		cEOF:	(*search for eof*)
			pInBuffer := ADR(InBuffer[0]); (*just for reference. Makes looking at data easier*)
			IF NOT DataAvailable THEN
				(*search buffer for EOF string*)
				FindState:=0; (*index for counting successive matches to EOF*)
				FOR index := 0 TO InBufferDataLength  + 1 DO
					IF InBuffer[index] = pEOF^[FindState] THEN
						(*match found*)
						FindState := FindState + 1;
						IF findState = EOFLength THEN
							EOFIndex:=index - EOFLength +1;
							EOFFound := TRUE;
							EXIT;
						END_IF
					ELSE
						IF FindState > 0 THEN
							FindState:=0; (*reset counter and start looking for new match*)
							IF InBuffer[index] = pEOF^[FindState] THEN (*must check current index for match to first element of EOF.*)
								FindState:=1;
							END_IF
						END_IF
					END_IF
				END_FOR;
			END_IF
			IF EOFFound THEN (*message found*)
				MEMCPY(pReceiveBuffer, ADR(InBuffer[0]),DINT_TO_UDINT(EOFIndex)); (*copy message up to but not including EOF into receive message*)
				Index := EOFIndex + EOFLength;
				ReceiveLength := EOFIndex ;
				IF ((Index ) < InBufferDataLength) THEN
					MEMSET(ADR(TempBuffer),0,SIZEOF(TempBuffer));
					MEMCPY(ADR(TempBuffer[0]),ADR(InBuffer[index]),DINT_TO_UDINT(InBufferDataLength-Index));
					MEMSET( ADR(InBuffer),0,SIZEOF(InBuffer));
					InBufferDataLength := InBufferDataLength-Index;
					MEMCPY(ADR(InBuffer[0]),ADR(TempBuffer[0]),DINT_TO_UDINT(InBufferDataLength));
					InBufferDataLength := 0;
				ELSE
					MEMSET( ADR(InBuffer),0,SIZEOF(InBuffer));
					InBufferDataLength := 0;
				END_IF
				EOFIndex := 0;
				EOFFound := FALSE;
				DataAvailable := 1;
			END_IF

			NextState := 0;

		cFixedLength:		(*fixed receive lengh*)
			IF NOT DataAvailable AND (InBufferDataLength >= FixedMessageLength) THEN
				MEMCPY(pReceiveBuffer, ADR(InBuffer[0]),DINT_TO_UDINT(FixedMessageLength)); (*copy data to output *)
				ReceiveLength := FixedMessageLength;
				InBufferDataLength := InBufferDataLength - FixedMessageLength;
				IF InBufferDataLength > 0 THEN
					(*still have data*)
					MEMCPY(ADR(TempBuffer[0]),ADR(InBuffer[FixedMessageLength]),DINT_TO_UDINT(InBufferDataLength));
					MEMSET( ADR(InBuffer),0,SIZEOF(InBuffer));
					MEMCPY(ADR(InBuffer[0]),ADR(TempBuffer[0]),DINT_TO_UDINT(InBufferDataLength));
				ELSE
					MEMSET( ADR(InBuffer),0,SIZEOF(InBuffer));
					InBufferDataLength := 0;
				END_IF
				DataAvailable := 1;
			END_IF
			NextState := 0;

		cContinuous:		(*continuous read*)
			IF NOT DataAvailable AND (InBufferDataLength <> PreviousInMessageLength) THEN
				PreviousInMessageLength := InBufferDataLength;
			ELSIF NOT DataAvailable AND (InBufferDataLength = PreviousInMessageLength) AND (InBufferDataLength > 0) THEN
				MEMCPY(pReceiveBuffer, ADR(InBuffer[0]),DINT_TO_UDINT(InBufferDataLength)); (*copy data to output *)
				ReceiveLength := InBufferDataLength;
				InBufferDataLength := 0;
				MEMSET( ADR(InBuffer),0,SIZEOF(InBuffer));
				DataAvailable := 1;
			END_IF
			NextState := 0;
			
		cVarSize:
			tmrReceive(PT:=T#300MS);
			IF NOT DataAvailable AND (InBufferDataLength <> PreviousInMessageLength) THEN
				tmrReceive(IN:=FALSE);
				PreviousInMessageLength := InBufferDataLength;
				tmrReceive(IN:=TRUE);
			ELSIF NOT DataAvailable AND (InBufferDataLength = PreviousInMessageLength) AND (InBufferDataLength > 0) AND tmrReceive.Q THEN
				tmrReceive(IN:=FALSE);
				MEMCPY(pReceiveBuffer, ADR(InBuffer[0]),DINT_TO_UDINT(InBufferDataLength)); (*copy data to output *)
				ReceiveLength := InBufferDataLength;
				InBufferDataLength := 0;
				MEMSET( ADR(InBuffer),0,SIZEOF(InBuffer));
				DataAvailable := 1;
			END_IF
			NextState := 0;
 
		ELSE
			(*Software error*)
			Error:=1;
			ErrorCode:=9;
			NextState := 0;
	END_CASE;

200:	(*Message read, clear output*)

	IF  FirstEntry THEN
		DataAvailable:=0;
		MEMSET(pReceiveBuffer,0,SIZEOF(pReceiveBuffer^));
		ReceiveLength:=0;
	END_IF
	IF NOT ReceiveData THEN
		NextState:=0;
	END_IF

END_CASE

(*set output device bits*)
LastSW := iRS232SW;

END_FUNCTION_BLOCK

// ---- POUs/State Trace/FIFO_StateTrace.TcPOU
FUNCTION_BLOCK FIFO_StateTrace
VAR_INPUT
	Overwrite	: BOOL;							// Flag to Overwrite FIFO Elements (when filled)
	pFIFO		: POINTER TO TraceFIFOBuffer;	// Pointer to FIFO Memory
END_VAR

VAR_OUTPUT
	Error		: BOOL;							// Flag Indicating Error with FIFO
	Count		: DINT;							// Count of Elements Within FIFO
	Full		: BOOL;							// Flag Indicating FIFO Full
END_VAR

VAR
	Head		: UDINT;						// Index of Head Element (Newest)
	Tail		: UDINT;						// Index of Tail Element (Oldest)
END_VAR

ACTION INIT:
// Clear Buffer and Output Data
MEMSET(ADR(pFIFO^.Buffer), 0, SIZEOF(pFIFO^.Buffer));

// Reset Count / Indicies
Count 	:= 0;
Head 	:= 0;
Tail 	:= 0;

// Reset Flags
Full 	:= FALSE;
Error 	:= FALSE;
END_ACTION

METHOD LOAD : BOOL
VAR_INPUT
	Input	: StatsEvent;
END_VAR
// Set Success Flag
Error := FALSE;
LOAD := TRUE;

// Check if FIFO Has Room (or Overwrite Enabled)
IF (Full AND Overwrite) OR NOT Full THEN
	
	// Set Head Element to Input Value
	pFIFO^.Buffer[Head] := Input;
	
	// Iterate Head Index
	Head := Head + 1;
	
	// Check if Head at Maximum Value, Rollover
	IF Head = pFIFO^.Size THEN
		Head := 0;
	END_IF
	
	// If FIFO Full, Iterate Tail
	IF Full THEN
		Tail := Tail + 1;
		
		// If Tail at Maximum Value, Rollover
		IF Tail = pFIFO^.Size THEN
			Tail := 0;
		END_IF
		
	// Otherwise Update Count
	ELSE
		Count := Count + 1;
	END_IF
	
// Otherwise, Flag Failure (Value Appended to Full FIFO)
ELSE
	Error := TRUE;
	LOAD := FALSE;
	
END_IF

Full := Head = Tail;
END_METHOD

METHOD PEEK : StatsEvent
// Reset Error Flag
Error := FALSE;

// Check if FIFO Full or Tail
IF Count > 0 THEN
	PEEK := pFIFO^.Buffer[Tail];
	
// Otherwise, Flag Error (FIFO is Empty)
ELSE
	Error := TRUE;
END_IF
END_METHOD

METHOD UNLOAD : StatsEvent
// Reset Error Flag
Error := FALSE;

// Check if FIFO Has Elements
IF Count > 0 THEN
	
	// Fetch Oldest Value from FIFO
	UNLOAD := pFIFO^.Buffer[Tail];
	
	// Clear FIFO Position
	pFIFO^.Buffer[Tail] := 0; 
	
	// Update Oldest Value Index
	Tail := Tail + 1;
	
	// Update Element Count
	Count := Count - 1;
	
	// Check for Rollover
	IF Tail = pFIFO^.Size THEN
		Tail := 0;
	END_IF
	
	// Reset Full Flag
	Full := FALSE;
	
// Otherwise, Flag Error (FIFO is Empty)
ELSE
	Error 	:= TRUE;
	UNLOAD := 0;
END_IF
END_METHOD

END_FUNCTION_BLOCK

// ---- POUs/TCP Communication/FB_TCPClient.TcPOU
// Function Block Organizing TCP Client Connection and Communication to Server
FUNCTION_BLOCK FB_TCPClient
// Inputs and Commands
VAR_INPUT
	RemoteHost			: STRING(15);				// Remote TCP Server Address
	RemotePort			: UDINT;					// Remote TCP Server Port
	Connect				: BOOL;						// Command to Connect Client to Remote Server
	Send				: BOOL;						// Command to Send TCP Message to Remote Server
	Received			: BOOL;						// Command to Indicate Message Received, Reset for Additional Receives 
	ClearError			: BOOL;						// Command to Clear Error Condition
	Flush				: BOOL;						// Command to Flush Buffers
	TransmitBuffer		: ARRAY [0..4095] OF BYTE;	// Buffer for TCP Message Send
	TransmitLength		: UDINT;					// Length of TCP Message
END_VAR

// Receive Configuration Inputs
VAR_INPUT
	MessageDelimiter	: ARRAY [0..11] OF BYTE;	// Buffer for TCP Message Delimiter
	DelimiterLength		: UDINT;					// Length of TCP Message Delimeter
	MessageLength		: UDINT;					// Fixed Length of TCP Messages
	ReceiveMode			: eRxMode;					// Message Receive Mode Configuration
END_VAR

// Outputs and Statuses
VAR_OUTPUT
	ReceiveBuffer		: ARRAY[0..4095] OF BYTE;	// Buffer Containing Received TCP Messages
	ReceiveLength		: UDINT;					// Length of Message in Receive Buffer
	DataAvailable		: BOOL;						// Flag Indicating New Receive Data Available
	Connected			: BOOL;						// Status of TCP Client Connection to Remote Server
	TransmitComplete	: BOOL;						// Flag Indicating TCP Message Send Completed
	Error				: BOOL;						// Flag Indicating Error with TCP Communication
	ErrorText			: T_MaxString;				// Human-Readable Text Related to Active Error Condition
	FlushComplete		: BOOL;						// Flag Indicating Flush of Buffers Complete
END_VAR

// Internal State Machine Variable
VAR
	State				: DINT;						// Current State of TCP Communications
	NextState			: DINT;						// Next State for TCP Communications
	FirstEntry			: BOOL;						// Flag Indicating First Entry to State
	StateDwellTimer		: TON;						// Timer for Dwell in States
	StateTimePreset		: TIME;						// Time Limit for Dwell in States
END_VAR

// Message Processing Variables
VAR
	RxBuffer			: ARRAY[0..4095] OF BYTE; 	// Buffer for Receiving Input Data
	InBuffer			: ARRAY[0..12287] OF BYTE;	// Buffer for Processing Input Data
	InBufferDataLength	: UDINT;					// Input Data Length
	TempBuffer			: ARRAY[0..12287] OF BYTE;	// Buffer for Bitwise Shifting of Messages
	Index				: UDINT;					// Index Used for Searching Buffers
	EOFIndex			: UDINT;					// Index of Delimiter
	EOFCount			: UDINT;					// Count of Delimiters 
END_VAR

// Low-Level TwinCAT TCP Libraries
VAR
	hSocketHandle		: T_HSOCKET;				// Handle for TCP Socket Connection
	fbSocketConnect		: FB_SocketConnect;			// Function Block for TCP Client Connection
	fbSocketClose		: FB_SocketClose;			// Function Block to Close TCP Socket
	fbSocketCloseAll	: FB_SocketCloseAll;		// Function Block to Close All Sockets
	fbSocketReceive		: FB_SocketReceive;			// Function Block to Poll Socket Memory Buffer
	fbSocketSend		: FB_SocketSend;			// Function Block to Send Message to Server
END_VAR

(*If State Change, capture rising edge with FirstEntry.*)
IF State <> NextState THEN
	FirstEntry := TRUE;
	State := NextState;
ELSE 
	FirstEntry := FALSE;
END_IF

StateDwellTimer(IN := State = NextState, PT := StateTimePreset);

(**********************
* Sequence logic *
***********************)
CASE State OF

0:	// Wait for Connect Command

	IF FirstEntry THEN
		fbSocketConnect(bExecute := FALSE);
		Connected := FALSE;
		DataAvailable := FALSE;
		FlushComplete := FALSE;
	END_IF
	
	IF Connect AND NOT Error THEN
		NextState := 100;
		
	ELSIF ClearError THEN
		Error := FALSE;
		ErrorText := '';
	END_IF
	

100:	// Validate TCP Server

	IF RemoteHost = '' OR RemotePort = 0 THEN
		Error := TRUE;
		ErrorText := 'Invalid connect parameters';
	END_IF
	
	IF NOT Error THEN
		NextState := 110;
	ELSE
		NextState := 0;
	END_IF

	
110:	// Connect to Server

	IF FirstEntry THEN
		fbSocketConnect(
			sSrvNetId 	:= '',
			sRemoteHost := RemoteHost,
			nRemotePort := RemotePort,
			bExecute 	:= TRUE,
			tTimeout 	:= T#15S);
	END_IF
	
	IF fbSocketConnect.bBusy THEN
		NextState := 120;
	END_IF

	
120:	// Wait for Connection

	StateTimePreset := T#4S;
	
	fbSocketConnect(bExecute:= FALSE);
	
	// Wait for Connect to Complete
	IF NOT fbSocketConnect.bBusy THEN
		// If Connected with Error
		IF fbSocketConnect.bError THEN
			Error := TRUE;
			ErrorText:= 'Socket Connection Could Not Be Made To ';
			ErrorText := CONCAT(ErrorText, RemoteHost);
			ErrorText := CONCAT(ErrorText, ' Port ');
 			ErrorText := CONCAT(ErrorText, TO_STRING(RemotePort));
			NextState := 500; // Error State
		ELSE
			// Check if Handle Created
			IF fbSocketConnect.hSocket.handle > 0 THEN
				hSocketHandle := fbSocketConnect.hSocket;
				Connected := TRUE;
				NextState := 600; // Clear Input Buffer
			ELSE
				Error := TRUE;
				ErrorText := 'Improper Handle Created by Connection ';
				ErrorText := CONCAT(ErrorText, TO_STRING(fbSocketConnect.hSocket.handle));
				NextState := 500;
			END_IF
		END_IF
	ELSE
		// Timeout After Preset
		IF StateDwellTimer.Q THEN
			Error := TRUE;
			ErrorText := 'Socket Connection Timed Out: ';
			ErrorText := CONCAT(ErrorText, RemoteHost);
			ErrorText := CONCAT(ErrorText, ' Port ');
 			ErrorText := CONCAT(ErrorText, TO_STRING(RemotePort));
			NextState := 500; // Error State
		END_IF
	END_IF

	
200: // Client Connected, Wait for Command

	// Connect Command Removed
	IF NOT Connect THEN
		NextState := 500;
	END_IF
	
	// Receive Message Command
	IF Received THEN
		NextState := 300;
	END_IF
	
	// Send Message Command
	IF Send THEN
		NextState := 400;
	END_IF
	
	// Flush Buffers Command
	IF Flush THEN
		NextState := 600;
	END_IF

	StateTimePreset := T#100MS;
	
	// Poll for New Receive
	IF StateDwellTimer.Q AND NextState = 200 THEN
		NextState := 210;
		fbSocketReceive(bExecute := FALSE);
	END_IF
	

210: 	// Poll Receive Buffer

	IF FirstEntry THEN
		fbSocketReceive(
			sSrvNetId 	:= '',
			hSocket 	:= hSocketHandle ,
			cbLen 		:= SIZEOF(RxBuffer),
			pDest 		:= ADR(RxBuffer),
			bExecute 	:= TRUE,
			tTimeout 	:= T#5S);
	END_IF
	
	IF NOT FirstEntry AND fbSocketReceive.bBusy THEN
		NextState := 220;
	END_IF
	

220:	// Wait for Return

	fbSocketReceive(bExecute := FALSE);
	
	IF NOT fbSocketReceive.bBusy THEN
		IF NOT fbSocketReceive.bError THEN
			IF fbSocketReceive.nRecBytes > 0 THEN
				NextState := 230;
			ELSE
				NextState := 200;
			END_IF
		ELSE
			Error := 1;
			ErrorText := 'Socket Receive Error: ';
			ErrorText := CONCAT(ErrorText, RemoteHost);
			ErrorText := CONCAT(ErrorText, ' Port ');
 			ErrorText := CONCAT(ErrorText, DINT_TO_STRING(RemotePort));
			NextState := 500;
		END_IF
	END_IF

	
230: // Copy Received Data

	// Check if Data Fits in Input Buffer
	IF (fbSocketReceive.nRecBytes + InBufferDataLength) <= SIZEOF(InBuffer) THEN
		
		// Copy Data from Receive Buffer to Input Buffer
		MEMCPY(ADR(InBuffer[InBufferDataLength]), ADR(RxBuffer), fbSocketReceive.nRecBytes);
		InBufferDataLength := InBufferDataLength + fbSocketReceive.nRecBytes;
		
		// Clear Receive Buffer
		MEMSET(ADR(RxBuffer), 0, SIZEOF(RxBuffer));
		NextState := 240;
	ELSE
		Error := 1;
		ErrorText := 'Buffer Overflow';
		NextState := 500;
	END_IF

	
240: // Construct TCP Message

	CASE ReceiveMode OF

		// Search for Delimiter
		eRxMode.Delimited:

			// Message Not Defined, Search Buffer
			IF NOT DataAvailable THEN
				
				// Initialize Delimiter Count
				EOFCount := 0;
				
				// Search Buffer from Tail
				FOR Index := 0 TO InBufferDataLength - 1 DO
					// If Match Found - Iterate EOF Count (For Delimiter Length)
					IF InBuffer[index] = MessageDelimiter[EOFCount] THEN
						EOFCount := EOFCount + 1;
						IF EOFCount = DelimiterLength THEN
							EOFIndex := Index - DelimiterLength + 1;
							EXIT;
						END_IF
					ELSE
						// If EOF Count > 0, Reset and Continue Search 
						IF EOFCount > 0 THEN
							EOFCount := 0;
							IF InBuffer[index] = MessageDelimiter[EOFCount] THEN
								EOFCount := 1;
							END_IF
						END_IF
					END_IF
				END_FOR;
			END_IF
			
			// Message Found in Buffer
			IF EOFIndex > 0 THEN 
				// Copy Message (Including Delimiter) to Receive Buffer
				ReceiveLength := EOFIndex + DelimiterLength;
				MEMCPY(ADR(ReceiveBuffer), ADR(InBuffer[0]), ReceiveLength);
				Index := EOFIndex + DelimiterLength;
				
				// If Data Remaining in Input Buffer, Bit-Shift to Head
				IF ReceiveLength < InBufferDataLength THEN
					MEMCPY(ADR(TempBuffer), ADR(InBuffer[ReceiveLength]), InBufferDataLength - ReceiveLength);
					MEMSET(ADR(InBuffer), 0, SIZEOF(InBuffer));
					InBufferDataLength := InBufferDataLength - ReceiveLength;
					MEMCPY(ADR(InBuffer), ADR(TempBuffer), InBufferDataLength);
					MEMSET(ADR(TempBuffer), 0, SIZEOF(TempBuffer));
					
				// Otherwise, Clear Input Buffer
				ELSE
					MEMSET(ADR(InBuffer), 0, SIZEOF(InBuffer));
					InBufferDataLength := 0;
				END_IF
				
				DataAvailable := TRUE;
				EOFIndex := 0;
			END_IF
			
			NextState := 200; // Return to Dispatch

			
		eRxMode.FixedLength: 

			
			IF NOT DataAvailable THEN
				// Check if Input Data Sufficient Length
				IF InBufferDataLength >= MessageLength THEN
					// Copy Message to Receive Buffer
					MEMCPY(ADR(ReceiveBuffer), ADR(InBuffer), MessageLength);
					ReceiveLength := MessageLength;
					InBufferDataLength := InBufferDataLength - MessageLength;
					
					// If Input Buffer Still Contains Data, Bit-Shift to Head
					IF InBufferDataLength > 0 THEN
						MEMCPY(ADR(TempBuffer), ADR(InBuffer[MessageLength]), InBufferDataLength);
						MEMSET(ADR(InBuffer), 0, SIZEOF(InBuffer));
						MEMCPY(ADR(InBuffer), ADR(TempBuffer), InBufferDataLength);
					
					// Otherwise, Clear Input Buffer
					ELSE
						MEMSET(ADR(InBuffer),0,SIZEOF(InBuffer));
						InBufferDataLength := 0;
					END_IF
					
					DataAvailable := TRUE;
				END_IF
			END_IF
			
			NextState := 200; // Return to Dispatch
			

		eRxMode.Continuous:
 
			NextState := 200; // Return to Dispatch
			
			
		ELSE
			Error := TRUE;
			ErrorText := 'Unknown RxMode Selected';
			NextState := 500;
			
	END_CASE;


300:	// Reset Message Received Buffer

	IF FirstEntry THEN
		DataAvailable := FALSE;
		MEMSET(ADR(ReceiveBuffer), 0, SIZEOF(ReceiveBuffer));
		ReceiveLength := 0;
	END_IF

	IF NOT Received THEN
		// If Data in Input Buffer, Process and Receive
		IF InBufferDataLength > 0 THEN
			NextState := 240; // Receive Data
		ELSE
			NextState := 200; // Dispatch
		END_IF
	END_IF
	

400:	// Transmit Data

	IF FirstEntry THEN
		fbSocketSend(bExecute := FALSE);
		fbSocketSend(
			sSrvNetId 	:= '',
			hSocket 	:= hSocketHandle,
			cbLen 		:= TransmitLength + 1,
			pSrc 		:= ADR(TransmitBuffer),
			bExecute 	:= TRUE,
			tTimeout 	:= T#5S);
	END_IF
	
	IF NOT FirstEntry THEN
		IF fbSocketSend.bBusy THEN
			TransmitComplete := TRUE;
			NextState := 410; // Wait for Reset
		ELSIF fbSocketSend.bError THEN
			Error := TRUE;
			ErrorText := 'TCP/IP Send error';
			NextState := 500; // Close TCP Connection
		END_IF
	END_IF

	
410:	// Wait for Send Reset

	fbSocketSend(bExecute := FALSE);
	
	IF NOT Send THEN
		TransmitComplete := FALSE;
		NextState := 200;
	END_IF

	
500:	// Close Connection

	IF FirstEntry THEN
		fbSocketClose(bExecute:= FALSE);
		fbSocketClose(
			sSrvNetId 	:= '',
			hSocket 	:= hSocketHandle,
			bExecute 	:= TRUE,
			tTimeout 	:= T#15S);
	END_IF
	
	StateTimePreset := T#1S;
	
	IF fbSocketClose.bBusy THEN
		NextState := 510;
	END_IF
	
	IF StateDwellTimer.Q THEN
		Error := TRUE;
		ErrorText := 'Socket Close Error: ';
		ErrorText := CONCAT(ErrorText, RemoteHost);
		ErrorText := CONCAT(ErrorText, ' Port ');
		ErrorText := CONCAT(ErrorText, DINT_TO_STRING(RemotePort));
		NextState := 510;
	END_IF

	
510: // Wait for Close

	fbSocketClose(bExecute := FALSE);
	
	IF NOT fbSocketClose.bBusy THEN
		NextState := 0;
	END_IF

	
600: 	// Clear Data from Buffers

	IF FirstEntry THEN
		MEMSET(ADR(InBuffer), 0, SIZEOF(InBuffer));
		MEMSET(ADR(TempBuffer), 0, SIZEOF(TempBuffer));
		MEMSET(ADR(ReceiveBuffer), 0, SIZEOF(ReceiveBuffer));
		InBufferDataLength := 0;
		Error := FALSE;
		DataAvailable := FALSE;
		TransmitComplete := FALSE;
		FlushComplete := TRUE;
	END_IF
	
	IF NOT Flush THEN
		FlushComplete := FALSE;
		NextState := 200;
	END_IF

END_CASE

END_FUNCTION_BLOCK

// ---- POUs/Utility/FB_FileReadSettings.TcPOU
FUNCTION_BLOCK FB_FileReadSettings
VAR_INPUT
	pReadData: POINTER TO BYTE;
	SizeOfData: DINT;
	FileName: T_MaxString; (* file path and name *)
	bExecute: BOOL; (* rising edge starts fb execution *)
END_VAR

VAR_OUTPUT
	bError: BOOL;
	bDone: BOOL;
END_VAR

VAR
	nErrId: UDINT;
	bBusy: BOOL;
	fbFileOpen: FB_FileOpen;
	fbFileClose: FB_FileClose;
	fbFileRead: FB_FileRead;

	hFile: UINT	:= 0; (* file handle of the file *)

	Step: DWORD;
	RisingEdge: R_TRIG;

	cbReadLength: UDINT := 0;
END_VAR


CASE Step OF
	
	0: (* do nothing *)
	;

	1: (* open file *)
	
	fbFileOpen(bExecute := FALSE);
	fbFileOpen(sNetId := '',
		sPathName := FileName,
		nMode := FOPEN_MODEREAD OR FOPEN_MODEBINARY,
		ePath := PATH_GENERIC,
		tTimeout := T#2s,
		bExecute := TRUE );
		Step := Step + 1;

	2:
	fbFileOpen(bExecute := FALSE);
	IF (NOT fbFileOpen.bBusy) THEN
		IF fbFileOpen.bError THEN
			nErrId := fbFileOpen.nErrId;
			bError := TRUE;
			Step := 50;
		ELSE
			hFile := fbFileOpen.hFile;
			Step := 5;
		END_IF
	END_IF

	5: (*read data from source file*)
	cbReadLength := 0;
	fbFileRead(bExecute := FALSE);
	fbFileRead(sNetId := '',
			hFile := hFile,
			pReadBuff := pReadData,
			cbReadLen := SizeOfData,
			bExecute := TRUE,
			tTimeout := T#2S);
	Step := Step + 1;

	6:
	fbFileRead(bExecute := FALSE);
	IF (NOT fbFileRead.bBusy) THEN
		IF fbFileRead.bError THEN
			nErrId := fbFileRead.nErrId;
			bError := TRUE;
			Step := 50;
		ELSIF fbFileRead.cbRead <> SizeOfData THEN
			nErrId := fbFileRead.nErrId;
			bError := TRUE;
			Step := 50;
		ELSE
			cbReadLength := fbFileRead.cbRead;
			Step := 50;
		END_IF
	END_IF


	30: (* close the file *)
	fbFileClose(bExecute := FALSE);
	fbFileClose(sNetId := '',
			hFile := hFile,
			bExecute := TRUE,
			tTimeout := T#2S);
	Step := Step + 1;

	31:
	fbFileClose(bExecute := FALSE);
	IF (NOT fbFileClose.bBusy) THEN
		IF fbFileClose.bError THEN
			nErrId := fbFileClose.nErrId;
			bError := TRUE;
		END_IF
		Step := 50;
		hFile := 0;
	END_IF


	50: (*error or ready => cleanup*)
	IF hFile <> 0 THEN
		Step := 30; (* close the file*)
	ELSE
		Step := 0;	(* ready *)
		bBusy := FALSE;
	END_IF

END_CASE

END_FUNCTION_BLOCK

// ---- POUs/Utility/FB_FileWriteSettings.TcPOU
FUNCTION_BLOCK FB_FileWriteSettings
VAR_INPUT
	DataToWrite		: BYTE;
	SizeOfData		: DINT;
	FileName		: T_MaxString; (* file path and name *)
	bExecute: BOOL; (* rising edge starts fb execution *)
END_VAR

VAR_OUTPUT
	bError: BOOL;
	bDone: BOOL;
END_VAR

VAR
	nErrId: UDINT;
	bBusy: BOOL;
	fbFileOpen: FB_FileOpen;
	fbFileClose: FB_FileClose;
	fbFileWrite: FB_FileWrite;

	hFile: UINT := 0; (* file handle of the file *)

	Step: DWORD;
	RisingEdge: R_TRIG;
END_VAR


	fbFileOpen(bExecute := FALSE);
	fbFileOpen(sNetId := '',
			sPathName := FileName,
			nMode := FOPEN_MODEWRITE OR FOPEN_MODEBINARY,
			ePath := PATH_GENERIC,
			tTimeout := T#2s,
			bExecute := TRUE);
	Step := Step + 1;

	4:
	fbFileOpen(bExecute := FALSE);
	IF (NOT fbFileOpen.bBusy) THEN
		IF fbFileOpen.bError THEN
			nErrId := fbFileOpen.nErrId;
			bError := TRUE;
			Step := 50;
		ELSE
			hFile := fbFileOpen.hFile;
			Step := 7;
		END_IF
	END_IF

	7:(*write data to file*)
	fbFileWrite(bExecute := FALSE);
	fbFileWrite(sNetId := '',
			hFile := hFile,
			pWriteBuff := pDataToWrite,
			cbWriteLen := SizeOfData,
			bExecute := TRUE,
			tTimeout := T#2S);
	Step := Step + 1;

	8:
	fbFileWrite(bExecute := FALSE);
	IF (NOT fbFileWrite.bBusy) THEN
		IF fbFileWrite.bError THEN
			nErrId := fbFileWrite.nErrId;
			bError := TRUE;
			Step := 50;
		ELSE
			Step := 50; (*cleanup: close the file *)
		END_IF
	END_IF

	30:(* close the file *)
	fbFileClose(bExecute := FALSE);
	fbFileClose(sNetId := '',
			hFile := hFile,
			bExecute := TRUE,
			tTimeout := T#2S);
	Step := Step + 1;

	31:
	fbFileClose(bExecute := FALSE);
	IF (NOT fbFileClose.bBusy) THEN
		IF fbFileClose.bError THEN
			nErrId := fbFileClose.nErrId;
			bError := TRUE;
		END_IF
		Step := 50;
		hFile := 0;
	END_IF

	50: (*error or ready => cleanup*)
	IF (hFile <> 0) THEN
		Step := 30; (* close the destination file*)
	ELSE
		Step := 0; (* ready *)
		bBusy := FALSE;
	END_IF

END_CASE

END_FUNCTION_BLOCK

// ---- POUs/Utility/FB_Sensor.TcPOU
// Function Block for Delayed Triggers of DIO
FUNCTION_BLOCK FB_Sensor
VAR_INPUT
	Reset			: BOOL;	// Reset Timers/Outputs
	Input			: BOOL;	// Input Status
	OnDelayTime		: TIME;	// Delay to Set On TRUE After Input TRUE
	OffDelayTime	: TIME;	// Delay to Set Off TRUE After Input FALSE
END_VAR

VAR_OUTPUT
	On				: BOOL;	// Status of Delayed Input TRUE
	Off				: BOOL;	// Status of Delayed Input FALSE
END_VAR

VAR
	On_TON			: TON;	// TON Delay for Input TRUE
	Off_TON			: TON;	// TON Delay for Input False
END_VAR


// If Reset Commanded, Reset All
IF Reset THEN
	On_TON(IN := FALSE);
	Off_TON(IN := FALSE);
	On := FALSE;
	Off := FALSE;
	
// Otherwise, Evaluate TONs Based on Input Status
ELSE
	On_TON(
		IN 	:= Input, 
		PT 	:= OnDelayTime,
		Q	=> On);
	
	Off_TON(
		IN 	:= NOT Input, 
		PT 	:= OffDelayTime,
		Q	=> Off);
END_IF;

END_FUNCTION_BLOCK

// ---- POUs/Utility/FIFO_DINT100.TcPOU
FUNCTION_BLOCK FIFO_DINT100
VAR_INPUT
	Overwrite	: BOOL;							// Flag to Overwrite FIFO Elements (when filled)
	pFIFO		: POINTER TO DINT100FIFOBuffer;	// Pointer to FIFO Memory
END_VAR

VAR_OUTPUT
	Error		: BOOL;							// Flag Indicating Error with FIFO
	Count		: DINT;							// Count of Elements Within FIFO
	Full		: BOOL;							// Flag Indicating FIFO Full
END_VAR

VAR
	Head		: UDINT;						// Index of Head Element (Newest)
	Tail		: UDINT;						// Index of Tail Element (Oldest)
END_VAR

ACTION INIT:
// Clear Buffer and Output Data
MEMSET(ADR(pFIFO^.Buffer), 0, SIZEOF(pFIFO^.Buffer));

// Reset Count / Indicies
Count 	:= 0;
Head 	:= 0;
Tail 	:= 0;

// Reset Flags
Full 	:= FALSE;
Error 	:= FALSE;
END_ACTION

METHOD LOAD : BOOL
VAR_INPUT
	Input	: DINT;
END_VAR
// Set Success Flag
Error := FALSE;
LOAD := TRUE;

// Check if FIFO Has Room (or Overwrite Enabled)
IF (Full AND Overwrite) OR NOT Full THEN
	
	// Set Head Element to Input Value
	pFIFO^.Buffer[Head] := Input;
	
	// Iterate Head Index
	Head := Head + 1;
	
	// Check if Head at Maximum Value, Rollover
	IF Head = pFIFO^.Size THEN
		Head := 0;
	END_IF
	
	// If FIFO Full, Iterate Tail
	IF Full THEN
		Tail := Tail + 1;
		
		// If Tail at Maximum Value, Rollover
		IF Tail = pFIFO^.Size THEN
			Tail := 0;
		END_IF
		
	// Otherwise Update Count
	ELSE
		Count := Count + 1;
	END_IF
	
// Otherwise, Flag Failure (Value Appended to Full FIFO)
ELSE
	Error := TRUE;
	LOAD := FALSE;
	
END_IF

Full := Head = Tail;
END_METHOD

METHOD PEEK : DINT
// Reset Error Flag
Error := FALSE;

// Check if FIFO Full or Tail
IF Count > 0 THEN
	PEEK := pFIFO^.Buffer[Tail];
	
// Otherwise, Flag Error (FIFO is Empty)
ELSE
	Error := TRUE;
END_IF
END_METHOD

METHOD UNLOAD : DINT
// Reset Error Flag
Error := FALSE;

// Check if FIFO Has Elements
IF Count > 0 THEN
	
	// Fetch Oldest Value from FIFO
	UNLOAD := pFIFO^.Buffer[Tail];
	
	// Clear FIFO Position
	pFIFO^.Buffer[Tail] := 0; 
	
	// Update Oldest Value Index
	Tail := Tail + 1;
	
	// Update Element Count
	Count := Count - 1;
	
	// Check for Rollover
	IF Tail = pFIFO^.Size THEN
		Tail := 0;
	END_IF
	
	// Reset Full Flag
	Full := FALSE;
	
// Otherwise, Flag Error (FIFO is Empty)
ELSE
	Error 	:= TRUE;
	UNLOAD := 0;
END_IF
END_METHOD

END_FUNCTION_BLOCK

// ---- POUs/Utility/FIFO_ID50.TcPOU
FUNCTION_BLOCK FIFO_ID50
VAR_INPUT
	Overwrite: BOOL;
	pFIFO: POINTER TO ID50FIFOBuffer;
	in: ComponentIdentifier;
END_VAR

VAR_OUTPUT
	Err: BOOL;
	Count: DINT;
	Full: BOOL;
	out: ComponentIdentifier;
END_VAR

VAR
	Head: UDINT;
	Tail: UDINT;
	Idx: UDINT;
END_VAR

ACTION INIT:
Idx := pFIFO^.Size * SIZEOF(in);
MEMSET(ADR(pFIFO^.Buffer[0]), 0, Idx);
MEMSET(ADR(in), 0, SIZEOF(in));
MEMSET(ADR(out), 0, SIZEOF(out));
Count := 0;
Head := 0;
Tail := 0;
Full := 0;
Err := 0;
END_ACTION

ACTION LOAD:
Err := 0;
IF (Full AND Overwrite) OR NOT Full THEN
	pFIFO^.Buffer[Head] := in;
	Head := Head + 1;
	IF Head = pFIFO^.Size THEN
		Head := 0;
	END_IF
	IF Full THEN
		Tail := Tail + 1;
		IF Tail = pFIFO^.Size THEN
			Tail := 0;
		END_IF
	ELSE
		Count := Count + 1;
	END_IF
ELSE
	Err := 1;
END_IF
Full := (Head = Tail);
END_ACTION

ACTION PEEK:
Err := 0;
IF Full OR (Tail <> Head) THEN
	out := pFIFO^.Buffer[Tail];
ELSE
	Err := 1; (*fifo is empty*)
END_IF
END_ACTION

ACTION UNLOAD:
Err := 0;
IF NOT Full AND (Head = Tail) THEN
	(*empty*)
	Err := 1;
ELSE
	out := pFIFO^.Buffer[Tail];
	MEMSET(ADR(pFIFO^.Buffer[Tail]), 0, SIZEOF (in));
	Tail := Tail + 1;
	Count := Count - 1;
	IF Tail = pFIFO^.Size THEN
		Tail := 0;
	END_IF
	Full := 0;
END_IF
END_ACTION

END_FUNCTION_BLOCK

// ---- POUs/Utility/FIFO_LREAL100.TcPOU
FUNCTION_BLOCK FIFO_LREAL100
VAR_INPUT
	Overwrite: BOOL;
	pFIFO: POINTER TO LREAL100FIFOBuffer;
	in: LREAL;
END_VAR

VAR_OUTPUT
	Err: BOOL;
	Count: DINT;
	Full: BOOL;
	out: LREAL;
END_VAR

VAR
	Head: UDINT;
	Tail: UDINT;
	Idx: UDINT;
END_VAR

ACTION INIT:
Idx := pFIFO^.Size * SIZEOF(in);
MEMSET(ADR(pFIFO^.Buffer[0]), 0, Idx);
MEMSET(ADR(in), 0, SIZEOF(in));
MEMSET(ADR(out), 0, SIZEOF(out));
Count := 0;
Head := 0;
Tail := 0;
Full := 0;
Err := 0;
END_ACTION

ACTION LOAD:
Err := 0;
IF (Full AND Overwrite) OR NOT Full THEN
	pFIFO^.Buffer[Head] := in;
	Head := Head + 1;
	IF Head = pFIFO^.Size THEN
		Head := 0;
	END_IF
	IF Full THEN
		Tail := Tail + 1;
		IF Tail = pFIFO^.Size THEN
			Tail := 0;
		END_IF
	ELSE
		Count := Count + 1;
	END_IF
ELSE
	Err := 1;
END_IF
Full := (Head = Tail);
END_ACTION

ACTION PEEK:
Err := 0;
IF Full OR (Tail <> Head) THEN
	out := pFIFO^.Buffer[Tail];
ELSE
	Err := 1; (*fifo is empty*)
END_IF
END_ACTION

ACTION UNLOAD:
Err := 0;
IF NOT Full AND (Head = Tail) THEN
	(*empty*)
	Err := 1;
ELSE
	out := pFIFO^.Buffer[Tail];
	MEMSET(ADR(pFIFO^.Buffer[Tail]), 0, SIZEOF (in));
	Tail := Tail + 1;
	Count := Count - 1;
	IF Tail = pFIFO^.Size THEN
		Tail := 0;
	END_IF
	Full := 0;
END_IF
END_ACTION

END_FUNCTION_BLOCK

// ---- POUs/Utility/LEFTBigString.TcPOU
FUNCTION LEFTBigString : BOOL

	VAR_INPUT
	pInputString: POINTER TO BYTE;
	SizeOfInputString: UINT;
	SizeToCopy: UINT;
	pOutputString: POINTER TO BYTE;
	SizeOfOutputString: UINT;
END_VAR

VAR
	i: INT;
	pOutputStringNull: POINTER TO BYTE;
END_VAR

(* Make sure output string is big enough to hold the characters *)
IF SizeOfOutputString < SizeToCopy THEN
	RETURN;
END_IF

(* Copy bytes from input string to output string *)
MEMCPY(pOutputString, pInputString, SizeToCopy);

(* Append null character to end of output string *)
pOutputStringNull := (pOutputString + UINT_TO_DINT(SizeToCopy));
pOutputStringNull^ := 0;
LEFTBigString := TRUE;

END_FUNCTION

// ---- POUs/Utility/RIGHTBigString.TcPOU
FUNCTION RIGHTBigString : BOOL
VAR_INPUT
	pInputString: POINTER TO BYTE;
	SizeOfInputString: UINT;
	SizeToCopy: UINT;
	pOutputString: POINTER TO BYTE;
	SizeOfOutputString: UINT;
END_VAR

VAR
	i: INT;
	pInputStringNull: POINTER TO BYTE;
	pOutputStringNull: POINTER TO BYTE;
	NumberOfInputStringCharacters: DINT;
END_VAR

(* Make sure output string is big enough to hold the characters *)
IF SizeOfOutputString < SizeToCopy THEN
	RETURN;
END_IF

(* Find address of null character for input string *)
pInputStringNull := pInputString;
FOR i := 0 TO SizeOfInputString DO
	IF pInputStringNull^ = 0 THEN
		EXIT;
	END_IF
	pInputStringNull := pInputStringNull + 1;
END_FOR

(* Check to see if there are enough characters in input string, otherwise copy them all *)
NumberOfInputStringCharacters := pInputStringNull - pInputString;
IF NumberOfInputStringCharacters < UINT_TO_DINT(SizeToCopy) THEN
	(* Copy bytes from input string to output string *)
	MEMCPY(pOutputString, pInputStringNull - NumberOfInputStringCharacters, NumberOfInputStringCharacters);

	(* Append null character to end of output string *)
	pOutputStringNull := (pOutputString + NumberOfInputStringCharacters);
	pOutputStringNull^ := 0;
	RETURN;
END_IF

(* Copy bytes from input string to output string *)
MEMCPY(pOutputString, pInputStringNull - UINT_TO_DINT(SizeToCopy), SizeToCopy);

(* Append null character to end of output string *)
pOutputStringNull := (pOutputString + UINT_TO_DINT(SizeToCopy));
pOutputStringNull^ := 0;

RIGHTBigString := TRUE;

END_FUNCTION
